LIN {X 0,Y 272.99,Z 560.234,A -85,B 0,C 180,E1 -18744.093,E2 -18744.093} C_VEL
LIN {X 0,Y 270.191,Z 556.625,A -85,B 0,C 180,E1 -18746.042,E2 -18746.042} C_VEL
LIN {X 0,Y 266.873,Z 552.939,A -85,B 0,C 180,E1 -18748.935,E2 -18748.935} C_VEL
LIN {X 0,Y 264.106,Z 550.779,A -85,B 0,C 180,E1 -18752.833,E2 -18752.833} C_VEL
LIN {X 0,Y 263.594,Z 550.284,A -85,B 0,C 180,E1 -18754.258,E2 -18754.258} C_VEL
LIN {X 0,Y 263.268,Z 551.296,A -85,B 0,C 180,E1 -18757.694,E2 -18757.694} C_VEL
LIN {X 0,Y 264.359,Z 553.676,A -85,B 0,C 180,E1 -18761.073,E2 -18761.073} C_VEL
LIN {X 0,Y 267.005,Z 559.232,A -85,B 0,C 180,E1 -18764.711,E2 -18764.711} C_VEL
LIN {X 0,Y 269.353,Z 563.234,A -85,B 0,C 180,E1 -18766.816,E2 -18766.816} C_VEL
LIN {X 0,Y 273.133,Z 570.637,A -85,B 0,C 180,E1 -18769.548,E2 -18769.548} C_VEL
LIN {X 0,Y 275.859,Z 576.586,A -85,B 0,C 180,E1 -18771.234,E2 -18771.234} C_VEL
LIN {X 0,Y 278.502,Z 582.767,A -85,B 0,C 180,E1 -18772.706,E2 -18772.706} C_VEL
LIN {X 0,Y 280.961,Z 589.169,A -85,B 0,C 180,E1 -18773.975,E2 -18773.975} C_VEL
LIN {X 0,Y 281.956,Z 602.893,A -85,B 0,C 180,E1 -18775.262,E2 -18775.262} C_VEL
LIN {X 0,Y 282.297,Z 616.005,A -85,B 0,C 180,E1 -18776.226,E2 -18776.226} C_VEL
LIN {X 0,Y 277.754,Z 659.548,A -85,B 0,C 180,E1 -18777.957,E2 -18777.957} C_VEL
LIN {X 0,Y 275.518,Z 672.942,A -85,B 0,C 180,E1 -18778.687,E2 -18778.687} C_VEL
LIN {X 0,Y 272.817,Z 685.651,A -85,B 0,C 180,E1 -18779.633,E2 -18779.633} C_VEL
LIN {X 0,Y 269.43,Z 698.811,A -85,B 0,C 180,E1 -18780.934,E2 -18780.934} C_VEL
LIN {X 0,Y 265.918,Z 710.541,A -85,B 0,C 180,E1 -18782.451,E2 -18782.451} C_VEL
LIN {X 0,Y 262.42,Z 721.186,A -85,B 0,C 180,E1 -18784.203,E2 -18784.203} C_VEL
LIN {X 0,Y 259.296,Z 730.12,A -85,B 0,C 180,E1 -18786.012,E2 -18786.012} C_VEL
LIN {X 0,Y 256.506,Z 737.614,A -85,B 0,C 180,E1 -18787.869,E2 -18787.869} C_VEL
LIN {X 0,Y 253.725,Z 745.099,A -85,B 0,C 180,E1 -18790.165,E2 -18790.165} C_VEL
LIN {X 0,Y 250.845,Z 753.157,A -85,B 0,C 180,E1 -18793.311,E2 -18793.311} C_VEL
LIN {X 0,Y 249.342,Z 760.427,A -85,B 0,C 180,E1 -18795.722,E2 -18795.722} C_VEL
LIN {X 0,Y 248.341,Z 765.333,A -85,B 0,C 180,E1 -18797.746,E2 -18797.746} C_VEL
LIN {X 0,Y 247.593,Z 770.085,A -85,B 0,C 180,E1 -18800.194,E2 -18800.194} C_VEL
LIN {X 0,Y 247.162,Z 773.704,A -85,B 0,C 180,E1 -18802.649,E2 -18802.649} C_VEL
LIN {X 0,Y 246.922,Z 776.292,A -85,B 0,C 180,E1 -18805.102,E2 -18805.102} C_VEL
LIN {X 0,Y 246.923,Z 777.505,A -85,B 0,C 180,E1 -18806.737,E2 -18806.737} C_VEL
LIN {X 0,Y 246.958,Z 778.268,A -85,B 0,C 180,E1 -18808.369,E2 -18808.369} C_VEL
LIN {X 0,Y 246.991,Z 778.625,A -85,B 0,C 180,E1 -18810,E2 -18810} C_VEL
LIN {X 0,Y 246.952,Z 778.591,A -85,B 0,C 180,E1 -18811.631,E2 -18811.631} C_VEL
LIN {X 0,Y 246.922,Z 778.159,A -85,B 0,C 180,E1 -18813.263,E2 -18813.263} C_VEL
LIN {X 0,Y 247.065,Z 776.008,A -85,B 0,C 180,E1 -18816.533,E2 -18816.533} C_VEL
LIN {X 0,Y 247.467,Z 773.301,A -85,B 0,C 180,E1 -18818.986,E2 -18818.986} C_VEL
LIN {X 0,Y 248.15,Z 769.569,A -85,B 0,C 180,E1 -18821.434,E2 -18821.434} C_VEL
LIN {X 0,Y 249.22,Z 764.704,A -85,B 0,C 180,E1 -18823.869,E2 -18823.869} C_VEL
LIN {X 0,Y 250.823,Z 758.565,A -85,B 0,C 180,E1 -18826.272,E2 -18826.272} C_VEL
LIN {X 0,Y 252.675,Z 751.27,A -85,B 0,C 180,E1 -18828.548,E2 -18828.548} C_VEL
LIN {X 0,Y 254.549,Z 743.052,A -85,B 0,C 180,E1 -18830.611,E2 -18830.611} C_VEL
LIN {X 0,Y 256.736,Z 733.463,A -85,B 0,C 180,E1 -18832.534,E2 -18832.534} C_VEL
LIN {X 0,Y 259.084,Z 722.81,A -85,B 0,C 180,E1 -18834.222,E2 -18834.222} C_VEL
LIN {X 0,Y 261.004,Z 712.424,A -85,B 0,C 180,E1 -18835.52,E2 -18835.52} C_VEL
LIN {X 0,Y 262.797,Z 701.051,A -85,B 0,C 180,E1 -18836.611,E2 -18836.611} C_VEL
LIN {X 0,Y 264.351,Z 688.267,A -85,B 0,C 180,E1 -18837.511,E2 -18837.511} C_VEL
LIN {X 0,Y 265.434,Z 675.829,A -85,B 0,C 180,E1 -18838.086,E2 -18838.086} C_VEL
LIN {X 0,Y 267.55,Z 612.058,A -85,B 0,C 180,E1 -18839.803,E2 -18839.803} C_VEL
LIN {X 0,Y 264.123,Z 582.382,A -85,B 0,C 180,E1 -18841.169,E2 -18841.169} C_VEL
LIN {X 0,Y 261.282,Z 564.651,A -85,B 0,C 180,E1 -18842.125,E2 -18842.125} C_VEL
LIN {X 0,Y 258.876,Z 558.576,A -85,B 0,C 180,E1 -18842.691,E2 -18842.691} C_VEL
LIN {X 0,Y 254.271,Z 541.842,A -85,B 0,C 180,E1 -18845.48,E2 -18845.48} C_VEL
LIN {X 0,Y 252.213,Z 535.351,A -85,B 0,C 180,E1 -18846.636,E2 -18846.636} C_VEL
LIN {X 0,Y 249.373,Z 529.876,A -85,B 0,C 180,E1 -18847.897,E2 -18847.897} C_VEL
LIN {X 0,Y 249.019,Z 528.423,A -85,B 0,C 180,E1 -18848.202,E2 -18848.202} C_VEL
LIN {X 0,Y 249.009,Z 528.461,A -85,B 0,C 180,E1 -18852.792,E2 -18852.792} C_VEL
LIN {X 0,Y 249.037,Z 528.454,A -85,B 0,C 180,E1 -18857.367,E2 -18857.367} C_VEL
LIN {X 0,Y 249.045,Z 528.46,A -85,B 0,C 180,E1 -18861.623,E2 -18861.623} C_VEL
LIN {X 0,Y 249.058,Z 528.461,A -85,B 0,C 180,E1 -18865.642,E2 -18865.642} C_VEL
LIN {X 0,Y 249.047,Z 528.44,A -85,B 0,C 180,E1 -18869.473,E2 -18869.473} C_VEL
LIN {X 0,Y 249.065,Z 528.458,A -85,B 0,C 180,E1 -18873.162,E2 -18873.162} C_VEL
LIN {X 0,Y 249.056,Z 528.434,A -85,B 0,C 180,E1 -18876.731,E2 -18876.731} C_VEL
LIN {X 0,Y 249.104,Z 528.453,A -85,B 0,C 180,E1 -18880.211,E2 -18880.211} C_VEL
LIN {X 0,Y 249.218,Z 528.409,A -85,B 0,C 180,E1 -18883.621,E2 -18883.621} C_VEL
LIN {X 0,Y 249.247,Z 528.434,A -85,B 0,C 180,E1 -18888.617,E2 -18888.617} C_VEL
LIN {X 0,Y 249.474,Z 528.375,A -85,B 0,C 180,E1 -18891.903,E2 -18891.903} C_VEL
LIN {X 0,Y 249.432,Z 528.412,A -85,B 0,C 180,E1 -18896.77,E2 -18896.77} C_VEL
LIN {X 0,Y 249.723,Z 528.342,A -85,B 0,C 180,E1 -18900,E2 -18900} C_VEL
LIN {X 0,Y 249.433,Z 528.41,A -85,B 0,C 180,E1 -18903.231,E2 -18903.231} C_VEL
LIN {X 0,Y 249.437,Z 528.393,A -85,B 0,C 180,E1 -18906.704,E2 -18906.704} C_VEL
LIN {X 0,Y 249.338,Z 528.401,A -85,B 0,C 180,E1 -18909.737,E2 -18909.737} C_VEL
LIN {X 0,Y 249.192,Z 528.424,A -85,B 0,C 180,E1 -18914.705,E2 -18914.705} C_VEL
LIN {X 0,Y 249.131,Z 528.438,A -85,B 0,C 180,E1 -18918.078,E2 -18918.078} C_VEL
LIN {X 0,Y 249.083,Z 528.449,A -85,B 0,C 180,E1 -18921.519,E2 -18921.519} C_VEL
LIN {X 0,Y 249.128,Z 528.446,A -85,B 0,C 180,E1 -18925.483,E2 -18925.483} C_VEL
LIN {X 0,Y 249.084,Z 528.44,A -85,B 0,C 180,E1 -18928.996,E2 -18928.996} C_VEL
LIN {X 0,Y 249.028,Z 528.466,A -85,B 0,C 180,E1 -18932.427,E2 -18932.427} C_VEL
LIN {X 0,Y 249.046,Z 528.46,A -85,B 0,C 180,E1 -18936.343,E2 -18936.343} C_VEL
LIN {X 0,Y 249.004,Z 528.464,A -85,B 0,C 180,E1 -18940.479,E2 -18940.479} C_VEL
LIN {X 0,Y 249.007,Z 528.47,A -85,B 0,C 180,E1 -18944.879,E2 -18944.879} C_VEL
LIN {X 0,Y 249.021,Z 528.511,A -85,B 0,C 180,E1 -18947.496,E2 -18947.496} C_VEL
LIN {X 0,Y 253.277,Z 541.471,A -85,B 0,C 180,E1 -18951.862,E2 -18951.862} C_VEL
LIN {X 0,Y 256.09,Z 551.518,A -85,B 0,C 180,E1 -18954.861,E2 -18954.861} C_VEL
LIN {X 0,Y 263.951,Z 568.494,A -85,B 0,C 180,E1 -18956.551,E2 -18956.551} C_VEL
LIN {X 0,Y 265.853,Z 573.462,A -85,B 0,C 180,E1 -18956.967,E2 -18956.967} C_VEL
LIN {X 0,Y 268.937,Z 591.166,A -85,B 0,C 180,E1 -18957.921,E2 -18957.921} C_VEL
LIN {X 0,Y 266.202,Z 662.562,A -85,B 0,C 180,E1 -18959.805,E2 -18959.805} C_VEL
LIN {X 0,Y 265.188,Z 675.566,A -85,B 0,C 180,E1 -18960.423,E2 -18960.423} C_VEL
LIN {X 0,Y 263.792,Z 688.171,A -85,B 0,C 180,E1 -18961.344,E2 -18961.344} C_VEL
LIN {X 0,Y 262.212,Z 699.557,A -85,B 0,C 180,E1 -18962.474,E2 -18962.474} C_VEL
LIN {X 0,Y 260.124,Z 711.119,A -85,B 0,C 180,E1 -18963.958,E2 -18963.958} C_VEL
LIN {X 0,Y 257.883,Z 721.5,A -85,B 0,C 180,E1 -18965.658,E2 -18965.658} C_VEL
LIN {X 0,Y 255.849,Z 729.998,A -85,B 0,C 180,E1 -18967.384,E2 -18967.384} C_VEL
LIN {X 0,Y 253.844,Z 737.814,A -85,B 0,C 180,E1 -18969.33,E2 -18969.33} C_VEL
LIN {X 0,Y 252.109,Z 744.593,A -85,B 0,C 180,E1 -18971.41,E2 -18971.41} C_VEL
LIN {X 0,Y 250.689,Z 750.647,A -85,B 0,C 180,E1 -18973.719,E2 -18973.719} C_VEL
LIN {X 0,Y 249.221,Z 755.677,A -85,B 0,C 180,E1 -18976.132,E2 -18976.132} C_VEL
LIN {X 0,Y 248.238,Z 759.549,A -85,B 0,C 180,E1 -18978.57,E2 -18978.57} C_VEL
LIN {X 0,Y 247.778,Z 761.529,A -85,B 0,C 180,E1 -18980.202,E2 -18980.202} C_VEL
LIN {X 0,Y 247.152,Z 764.272,A -85,B 0,C 180,E1 -18983.469,E2 -18983.469} C_VEL
LIN {X 0,Y 246.973,Z 765.002,A -85,B 0,C 180,E1 -18985.103,E2 -18985.103} C_VEL
LIN {X 0,Y 246.947,Z 765.341,A -85,B 0,C 180,E1 -18986.737,E2 -18986.737} C_VEL
LIN {X 0,Y 246.95,Z 765.302,A -85,B 0,C 180,E1 -18988.369,E2 -18988.369} C_VEL
LIN {X 0,Y 246.99,Z 764.874,A -85,B 0,C 180,E1 -18990,E2 -18990} C_VEL
LIN {X 0,Y 247.302,Z 762.765,A -85,B 0,C 180,E1 -18993.258,E2 -18993.258} C_VEL
LIN {X 0,Y 247.748,Z 760.11,A -85,B 0,C 180,E1 -18995.698,E2 -18995.698} C_VEL
LIN {X 0,Y 248.364,Z 756.449,A -85,B 0,C 180,E1 -18998.134,E2 -18998.134} C_VEL
LIN {X 0,Y 249.333,Z 751.675,A -85,B 0,C 180,E1 -19000.557,E2 -19000.557} C_VEL
LIN {X 0,Y 250.677,Z 745.646,A -85,B 0,C 180,E1 -19002.961,E2 -19002.961} C_VEL
LIN {X 0,Y 252.37,Z 738.111,A -85,B 0,C 180,E1 -19005.34,E2 -19005.34} C_VEL
LIN {X 0,Y 254.433,Z 728.656,A -85,B 0,C 180,E1 -19007.688,E2 -19007.688} C_VEL
LIN {X 0,Y 256.4,Z 718.895,A -85,B 0,C 180,E1 -19009.619,E2 -19009.619} C_VEL
LIN {X 0,Y 258.19,Z 709.249,A -85,B 0,C 180,E1 -19011.141,E2 -19011.141} C_VEL
LIN {X 0,Y 259.587,Z 700.508,A -85,B 0,C 180,E1 -19012.273,E2 -19012.273} C_VEL
LIN {X 0,Y 261.132,Z 689.591,A -85,B 0,C 180,E1 -19013.389,E2 -19013.389} C_VEL
LIN {X 0,Y 262.399,Z 676.059,A -85,B 0,C 180,E1 -19014.429,E2 -19014.429} C_VEL
LIN {X 0,Y 263.298,Z 663.443,A -85,B 0,C 180,E1 -19015.065,E2 -19015.065} C_VEL
LIN {X 0,Y 265.187,Z 610.796,A -85,B 0,C 180,E1 -19016.491,E2 -19016.491} C_VEL
LIN {X 0,Y 265.831,Z 588.852,A -85,B 0,C 180,E1 -19017.077,E2 -19017.077} C_VEL
LIN {X 0,Y 262.181,Z 567.297,A -85,B 0,C 180,E1 -19018.169,E2 -19018.169} C_VEL
LIN {X 0,Y 255.508,Z 551.152,A -85,B 0,C 180,E1 -19019.537,E2 -19019.537} C_VEL
LIN {X 0,Y 252.819,Z 540.961,A -85,B 0,C 180,E1 -19022.482,E2 -19022.482} C_VEL
LIN {X 0,Y 249.116,Z 528.446,A -85,B 0,C 180,E1 -19026.455,E2 -19026.455} C_VEL
LIN {X 0,Y 249.078,Z 528.446,A -85,B 0,C 180,E1 -19030.463,E2 -19030.463} C_VEL
LIN {X 0,Y 249.019,Z 528.448,A -85,B 0,C 180,E1 -19034.874,E2 -19034.874} C_VEL
LIN {X 0,Y 249.053,Z 528.465,A -85,B 0,C 180,E1 -19036.704,E2 -19036.704} C_VEL
LIN {X 0,Y 259.215,Z 557.612,A -85,B 0,C 180,E1 -19038.571,E2 -19038.571} C_VEL
LIN {X 0,Y 256.382,Z 625.461,A -85,B 0,C 180,E1 -19041.166,E2 -19041.166} C_VEL
LIN {X 0,Y 255.738,Z 638.323,A -85,B 0,C 180,E1 -19041.93,E2 -19041.93} C_VEL
LIN {X 0,Y 254.756,Z 651.647,A -85,B 0,C 180,E1 -19043.031,E2 -19043.031} C_VEL
LIN {X 0,Y 253.633,Z 664.149,A -85,B 0,C 180,E1 -19044.415,E2 -19044.415} C_VEL
LIN {X 0,Y 252.346,Z 676.451,A -85,B 0,C 180,E1 -19046.15,E2 -19046.15} C_VEL
LIN {X 0,Y 251.19,Z 687.217,A -85,B 0,C 180,E1 -19048.072,E2 -19048.072} C_VEL
LIN {X 0,Y 250.005,Z 691.571,A -85,B 0,C 180,E1 -19048.949,E2 -19048.949} C_VEL
LIN {X 0,Y 246.343,Z 698.223,A -85,B 0,C 180,E1 -19050.431,E2 -19050.431} C_VEL
LIN {X 0,Y 242.767,Z 704.382,A -85,B 0,C 180,E1 -19052.06,E2 -19052.06} C_VEL
LIN {X 0,Y 241.73,Z 707.892,A -85,B 0,C 180,E1 -19053.148,E2 -19053.148} C_VEL
LIN {X 0,Y 241.207,Z 713.595,A -85,B 0,C 180,E1 -19055.206,E2 -19055.206} C_VEL
LIN {X 0,Y 240.618,Z 719.237,A -85,B 0,C 180,E1 -19057.684,E2 -19057.684} C_VEL
LIN {X 0,Y 240.293,Z 723.943,A -85,B 0,C 180,E1 -19060.345,E2 -19060.345} C_VEL
LIN {X 0,Y 240.205,Z 727.388,A -85,B 0,C 180,E1 -19062.987,E2 -19062.987} C_VEL
LIN {X 0,Y 240.325,Z 729.1,A -85,B 0,C 180,E1 -19064.801,E2 -19064.801} C_VEL
LIN {X 0,Y 240.548,Z 730.266,A -85,B 0,C 180,E1 -19066.483,E2 -19066.483} C_VEL
LIN {X 0,Y 240.898,Z 731.008,A -85,B 0,C 180,E1 -19068.216,E2 -19068.216} C_VEL
LIN {X 0,Y 241.855,Z 731.244,A -85,B 0,C 180,E1 -19071.105,E2 -19071.105} C_VEL
LIN {X 0,Y 242.816,Z 730.604,A -85,B 0,C 180,E1 -19073.351,E2 -19073.351} C_VEL
LIN {X 0,Y 243.776,Z 729.566,A -85,B 0,C 180,E1 -19075.038,E2 -19075.038} C_VEL
LIN {X 0,Y 246.085,Z 726.341,A -85,B 0,C 180,E1 -19078.28,E2 -19078.28} C_VEL
LIN {X 0,Y 248.337,Z 722.512,A -85,B 0,C 180,E1 -19080.81,E2 -19080.81} C_VEL
LIN {X 0,Y 250.903,Z 717.616,A -85,B 0,C 180,E1 -19083.211,E2 -19083.211} C_VEL
LIN {X 0,Y 253.556,Z 712.049,A -85,B 0,C 180,E1 -19085.347,E2 -19085.347} C_VEL
LIN {X 0,Y 256.664,Z 705.116,A -85,B 0,C 180,E1 -19087.473,E2 -19087.473} C_VEL
LIN {X 0,Y 260.263,Z 695.935,A -85,B 0,C 180,E1 -19089.716,E2 -19089.716} C_VEL
LIN {X 0,Y 263.627,Z 686.39,A -85,B 0,C 180,E1 -19091.533,E2 -19091.533} C_VEL
LIN {X 0,Y 266.924,Z 675.627,A -85,B 0,C 180,E1 -19093.185,E2 -19093.185} C_VEL
LIN {X 0,Y 270.017,Z 663.83,A -85,B 0,C 180,E1 -19094.6,E2 -19094.6} C_VEL
LIN {X 0,Y 272.46,Z 651.925,A -85,B 0,C 180,E1 -19095.714,E2 -19095.714} C_VEL
LIN {X 0,Y 274.515,Z 638.818,A -85,B 0,C 180,E1 -19096.643,E2 -19096.643} C_VEL
LIN {X 0,Y 276.515,Z 620.559,A -85,B 0,C 180,E1 -19097.519,E2 -19097.519} C_VEL
LIN {X 0,Y 280.862,Z 583.373,A -85,B 0,C 180,E1 -19098.983,E2 -19098.983} C_VEL
LIN {X 0,Y 277.859,Z 577.693,A -85,B 0,C 180,E1 -19100.43,E2 -19100.43} C_VEL
LIN {X 0,Y 274.432,Z 572.112,A -85,B 0,C 180,E1 -19102.221,E2 -19102.221} C_VEL
LIN {X 0,Y 271.179,Z 567.198,A -85,B 0,C 180,E1 -19104.186,E2 -19104.186} C_VEL
LIN {X 0,Y 268.152,Z 563.271,A -85,B 0,C 180,E1 -19106.357,E2 -19106.357} C_VEL
LIN {X 0,Y 265.242,Z 559.819,A -85,B 0,C 180,E1 -19109.03,E2 -19109.03} C_VEL
LIN {X 0,Y 262.508,Z 557.611,A -85,B 0,C 180,E1 -19113.059,E2 -19113.059} C_VEL
LIN {X 0,Y 262.098,Z 557.203,A -85,B 0,C 180,E1 -19114.27,E2 -19114.27} C_VEL
LIN {X 0,Y 261.741,Z 558.144,A -85,B 0,C 180,E1 -19117.454,E2 -19117.454} C_VEL
LIN {X 0,Y 262.545,Z 560.201,A -85,B 0,C 180,E1 -19120.455,E2 -19120.455} C_VEL
LIN {X 0,Y 263.676,Z 562.983,A -85,B 0,C 180,E1 -19122.571,E2 -19122.571} C_VEL
LIN {X 0,Y 266.928,Z 569.26,A -85,B 0,C 180,E1 -19126.2,E2 -19126.2} C_VEL
LIN {X 0,Y 270.377,Z 576.507,A -85,B 0,C 180,E1 -19128.921,E2 -19128.921} C_VEL
LIN {X 0,Y 273.124,Z 582.914,A -85,B 0,C 180,E1 -19130.764,E2 -19130.764} C_VEL
LIN {X 0,Y 276.12,Z 590.349,A -85,B 0,C 180,E1 -19132.51,E2 -19132.51} C_VEL
LIN {X 0,Y 277.009,Z 593.418,A -85,B 0,C 180,E1 -19133.072,E2 -19133.072} C_VEL
LIN {X 0,Y 277.845,Z 607.865,A -85,B 0,C 180,E1 -19134.425,E2 -19134.425} C_VEL
LIN {X 0,Y 277.751,Z 618.425,A -85,B 0,C 180,E1 -19135.169,E2 -19135.169} C_VEL
LIN {X 0,Y 273.212,Z 659.053,A -85,B 0,C 180,E1 -19136.81,E2 -19136.81} C_VEL
LIN {X 0,Y 270.87,Z 672.342,A -85,B 0,C 180,E1 -19137.538,E2 -19137.538} C_VEL
LIN {X 0,Y 268.261,Z 683.948,A -85,B 0,C 180,E1 -19138.402,E2 -19138.402} C_VEL
LIN {X 0,Y 264.647,Z 697.137,A -85,B 0,C 180,E1 -19139.698,E2 -19139.698} C_VEL
LIN {X 0,Y 260.928,Z 709.059,A -85,B 0,C 180,E1 -19141.22,E2 -19141.22} C_VEL
LIN {X 0,Y 257.566,Z 718.845,A -85,B 0,C 180,E1 -19142.804,E2 -19142.804} C_VEL
LIN {X 0,Y 253.548,Z 729.603,A -85,B 0,C 180,E1 -19144.995,E2 -19144.995} C_VEL
LIN {X 0,Y 249.998,Z 738.361,A -85,B 0,C 180,E1 -19147.261,E2 -19147.261} C_VEL
LIN {X 0,Y 246.656,Z 746.661,A -85,B 0,C 180,E1 -19150.007,E2 -19150.007} C_VEL
LIN {X 0,Y 244.02,Z 753.185,A -85,B 0,C 180,E1 -19152.83,E2 -19152.83} C_VEL
LIN {X 0,Y 241.954,Z 762.239,A -85,B 0,C 180,E1 -19156.135,E2 -19156.135} C_VEL
LIN {X 0,Y 240.799,Z 768.416,A -85,B 0,C 180,E1 -19159.064,E2 -19159.064} C_VEL
LIN {X 0,Y 240.212,Z 772.409,A -85,B 0,C 180,E1 -19161.588,E2 -19161.588} C_VEL
LIN {X 0,Y 239.996,Z 774.455,A -85,B 0,C 180,E1 -19163.273,E2 -19163.273} C_VEL
LIN {X 0,Y 239.839,Z 776.177,A -85,B 0,C 180,E1 -19165.071,E2 -19165.071} C_VEL
LIN {X 0,Y 239.824,Z 777.297,A -85,B 0,C 180,E1 -19166.64,E2 -19166.64} C_VEL
LIN {X 0,Y 239.867,Z 778.07,A -85,B 0,C 180,E1 -19168.321,E2 -19168.321} C_VEL
LIN {X 0,Y 239.9,Z 778.432,A -85,B 0,C 180,E1 -19170,E2 -19170} C_VEL
LIN {X 0,Y 239.862,Z 778.402,A -85,B 0,C 180,E1 -19171.679,E2 -19171.679} C_VEL
LIN {X 0,Y 239.824,Z 777.978,A -85,B 0,C 180,E1 -19173.36,E2 -19173.36} C_VEL
LIN {X 0,Y 239.844,Z 777.109,A -85,B 0,C 180,E1 -19175.043,E2 -19175.043} C_VEL
LIN {X 0,Y 239.989,Z 775.839,A -85,B 0,C 180,E1 -19176.727,E2 -19176.727} C_VEL
LIN {X 0,Y 240.423,Z 773.143,A -85,B 0,C 180,E1 -19179.252,E2 -19179.252} C_VEL
LIN {X 0,Y 241.167,Z 769.423,A -85,B 0,C 180,E1 -19181.77,E2 -19181.77} C_VEL
LIN {X 0,Y 242.301,Z 764.57,A -85,B 0,C 180,E1 -19184.273,E2 -19184.273} C_VEL
LIN {X 0,Y 243.983,Z 758.445,A -85,B 0,C 180,E1 -19186.741,E2 -19186.741} C_VEL
LIN {X 0,Y 245.851,Z 751.48,A -85,B 0,C 180,E1 -19188.985,E2 -19188.985} C_VEL
LIN {X 0,Y 247.885,Z 742.978,A -85,B 0,C 180,E1 -19191.191,E2 -19191.191} C_VEL
LIN {X 0,Y 250.201,Z 733.413,A -85,B 0,C 180,E1 -19193.156,E2 -19193.156} C_VEL
LIN {X 0,Y 252.61,Z 722.793,A -85,B 0,C 180,E1 -19194.884,E2 -19194.884} C_VEL
LIN {X 0,Y 254.621,Z 712.468,A -85,B 0,C 180,E1 -19196.207,E2 -19196.207} C_VEL
LIN {X 0,Y 256.627,Z 700.06,A -85,B 0,C 180,E1 -19197.414,E2 -19197.414} C_VEL
LIN {X 0,Y 258.289,Z 686.996,A -85,B 0,C 180,E1 -19198.324,E2 -19198.324} C_VEL
LIN {X 0,Y 259.349,Z 673.611,A -85,B 0,C 180,E1 -19198.916,E2 -19198.916} C_VEL
LIN {X 0,Y 261.477,Z 613.223,A -85,B 0,C 180,E1 -19200.557,E2 -19200.557} C_VEL
LIN {X 0,Y 258.243,Z 584.392,A -85,B 0,C 180,E1 -19201.923,E2 -19201.923} C_VEL
LIN {X 0,Y 255.65,Z 567.616,A -85,B 0,C 180,E1 -19202.849,E2 -19202.849} C_VEL
LIN {X 0,Y 252.033,Z 558.209,A -85,B 0,C 180,E1 -19203.763,E2 -19203.763} C_VEL
LIN {X 0,Y 247.176,Z 540.889,A -85,B 0,C 180,E1 -19206.845,E2 -19206.845} C_VEL
LIN {X 0,Y 245.96,Z 537.781,A -85,B 0,C 180,E1 -19207.469,E2 -19207.469} C_VEL
LIN {X 0,Y 242.282,Z 530.723,A -85,B 0,C 180,E1 -19209.207,E2 -19209.207} C_VEL
LIN {X 0,Y 241.943,Z 529.312,A -85,B 0,C 180,E1 -19209.533,E2 -19209.533} C_VEL
LIN {X 0,Y 241.935,Z 529.338,A -85,B 0,C 180,E1 -19213.429,E2 -19213.429} C_VEL
LIN {X 0,Y 241.973,Z 529.343,A -85,B 0,C 180,E1 -19216.56,E2 -19216.56} C_VEL
LIN {X 0,Y 241.978,Z 529.344,A -85,B 0,C 180,E1 -19220.285,E2 -19220.285} C_VEL
LIN {X 0,Y 242.033,Z 529.323,A -85,B 0,C 180,E1 -19224.497,E2 -19224.497} C_VEL
LIN {X 0,Y 241.971,Z 529.324,A -85,B 0,C 180,E1 -19228.48,E2 -19228.48} C_VEL
LIN {X 0,Y 242.003,Z 529.339,A -85,B 0,C 180,E1 -19232.312,E2 -19232.312} C_VEL
LIN {X 0,Y 242.036,Z 529.306,A -85,B 0,C 180,E1 -19236.014,E2 -19236.014} C_VEL
LIN {X 0,Y 242.031,Z 529.336,A -85,B 0,C 180,E1 -19239.608,E2 -19239.608} C_VEL
LIN {X 0,Y 242.158,Z 529.288,A -85,B 0,C 180,E1 -19243.278,E2 -19243.278} C_VEL
LIN {X 0,Y 242.181,Z 529.317,A -85,B 0,C 180,E1 -19248.28,E2 -19248.28} C_VEL
LIN {X 0,Y 242.421,Z 529.253,A -85,B 0,C 180,E1 -19251.666,E2 -19251.666} C_VEL
LIN {X 0,Y 242.256,Z 529.305,A -85,B 0,C 180,E1 -19255.007,E2 -19255.007} C_VEL
LIN {X 0,Y 242.632,Z 529.238,A -85,B 0,C 180,E1 -19258.341,E2 -19258.341} C_VEL
LIN {X 0,Y 242.632,Z 529.236,A -85,B 0,C 180,E1 -19261.66,E2 -19261.66} C_VEL
LIN {X 0,Y 242.418,Z 529.267,A -85,B 0,C 180,E1 -19266.676,E2 -19266.676} C_VEL
LIN {X 0,Y 242.263,Z 529.286,A -85,B 0,C 180,E1 -19270.024,E2 -19270.024} C_VEL
LIN {X 0,Y 242.152,Z 529.296,A -85,B 0,C 180,E1 -19275.142,E2 -19275.142} C_VEL
LIN {X 0,Y 242.067,Z 529.326,A -85,B 0,C 180,E1 -19278.625,E2 -19278.625} C_VEL
LIN {X 0,Y 242.009,Z 529.32,A -85,B 0,C 180,E1 -19282.181,E2 -19282.181} C_VEL
LIN {X 0,Y 242.064,Z 529.331,A -85,B 0,C 180,E1 -19285.839,E2 -19285.839} C_VEL
LIN {X 0,Y 242.029,Z 529.317,A -85,B 0,C 180,E1 -19289.581,E2 -19289.581} C_VEL
LIN {X 0,Y 241.978,Z 529.338,A -85,B 0,C 180,E1 -19293.494,E2 -19293.494} C_VEL
LIN {X 0,Y 241.988,Z 529.346,A -85,B 0,C 180,E1 -19297.583,E2 -19297.583} C_VEL
LIN {X 0,Y 241.938,Z 529.355,A -85,B 0,C 180,E1 -19301.923,E2 -19301.923} C_VEL
LIN {X 0,Y 241.953,Z 529.487,A -85,B 0,C 180,E1 -19306.339,E2 -19306.339} C_VEL
LIN {X 0,Y 245.448,Z 539.786,A -85,B 0,C 180,E1 -19309.991,E2 -19309.991} C_VEL
LIN {X 0,Y 248.246,Z 548.984,A -85,B 0,C 180,E1 -19312.988,E2 -19312.988} C_VEL
LIN {X 0,Y 249.025,Z 551.686,A -85,B 0,C 180,E1 -19313.757,E2 -19313.757} C_VEL
LIN {X 0,Y 256.527,Z 567.423,A -85,B 0,C 180,E1 -19315.454,E2 -19315.454} C_VEL
LIN {X 0,Y 260.054,Z 575.918,A -85,B 0,C 180,E1 -19316.242,E2 -19316.242} C_VEL
LIN {X 0,Y 262.837,Z 592.295,A -85,B 0,C 180,E1 -19317.151,E2 -19317.151} C_VEL
LIN {X 0,Y 260.022,Z 663.023,A -85,B 0,C 180,E1 -19319.058,E2 -19319.058} C_VEL
LIN {X 0,Y 258.944,Z 676.006,A -85,B 0,C 180,E1 -19319.692,E2 -19319.692} C_VEL
LIN {X 0,Y 257.595,Z 688.014,A -85,B 0,C 180,E1 -19320.588,E2 -19320.588} C_VEL
LIN {X 0,Y 255.92,Z 699.316,A -85,B 0,C 180,E1 -19321.717,E2 -19321.717} C_VEL
LIN {X 0,Y 254.04,Z 709.803,A -85,B 0,C 180,E1 -19323.063,E2 -19323.063} C_VEL
LIN {X 0,Y 251.675,Z 720.483,A -85,B 0,C 180,E1 -19324.796,E2 -19324.796} C_VEL
LIN {X 0,Y 249.285,Z 730.052,A -85,B 0,C 180,E1 -19326.754,E2 -19326.754} C_VEL
LIN {X 0,Y 247.191,Z 737.892,A -85,B 0,C 180,E1 -19328.747,E2 -19328.747} C_VEL
LIN {X 0,Y 245.256,Z 745.115,A -85,B 0,C 180,E1 -19331.023,E2 -19331.023} C_VEL
LIN {X 0,Y 243.852,Z 750.763,A -85,B 0,C 180,E1 -19333.25,E2 -19333.25} C_VEL
LIN {X 0,Y 242.3,Z 755.813,A -85,B 0,C 180,E1 -19335.727,E2 -19335.727} C_VEL
LIN {X 0,Y 241.245,Z 759.7,A -85,B 0,C 180,E1 -19338.234,E2 -19338.234} C_VEL
LIN {X 0,Y 240.745,Z 761.688,A -85,B 0,C 180,E1 -19339.913,E2 -19339.913} C_VEL
LIN {X 0,Y 240.36,Z 763.265,A -85,B 0,C 180,E1 -19341.594,E2 -19341.594} C_VEL
LIN {X 0,Y 240.076,Z 764.444,A -85,B 0,C 180,E1 -19343.276,E2 -19343.276} C_VEL
LIN {X 0,Y 239.85,Z 765.529,A -85,B 0,C 180,E1 -19346.64,E2 -19346.64} C_VEL
LIN {X 0,Y 239.862,Z 765.495,A -85,B 0,C 180,E1 -19348.321,E2 -19348.321} C_VEL
LIN {X 0,Y 239.898,Z 765.077,A -85,B 0,C 180,E1 -19350,E2 -19350} C_VEL
LIN {X 0,Y 240.224,Z 762.982,A -85,B 0,C 180,E1 -19353.354,E2 -19353.354} C_VEL
LIN {X 0,Y 240.699,Z 760.34,A -85,B 0,C 180,E1 -19355.865,E2 -19355.865} C_VEL
LIN {X 0,Y 241.337,Z 756.692,A -85,B 0,C 180,E1 -19358.372,E2 -19358.372} C_VEL
LIN {X 0,Y 242.367,Z 751.93,A -85,B 0,C 180,E1 -19360.864,E2 -19360.864} C_VEL
LIN {X 0,Y 243.762,Z 745.917,A -85,B 0,C 180,E1 -19363.335,E2 -19363.335} C_VEL
LIN {X 0,Y 245.549,Z 738.406,A -85,B 0,C 180,E1 -19365.777,E2 -19365.777} C_VEL
LIN {X 0,Y 247.684,Z 728.971,A -85,B 0,C 180,E1 -19368.187,E2 -19368.187} C_VEL
LIN {X 0,Y 249.742,Z 719.241,A -85,B 0,C 180,E1 -19370.165,E2 -19370.165} C_VEL
LIN {X 0,Y 251.858,Z 708.257,A -85,B 0,C 180,E1 -19371.914,E2 -19371.914} C_VEL
LIN {X 0,Y 253.502,Z 697.557,A -85,B 0,C 180,E1 -19373.269,E2 -19373.269} C_VEL
LIN {X 0,Y 255.139,Z 685.78,A -85,B 0,C 180,E1 -19374.404,E2 -19374.404} C_VEL
LIN {X 0,Y 256.275,Z 673.355,A -85,B 0,C 180,E1 -19375.282,E2 -19375.282} C_VEL
LIN {X 0,Y 257.092,Z 660.341,A -85,B 0,C 180,E1 -19375.879,E2 -19375.879} C_VEL
LIN {X 0,Y 259.568,Z 589.737,A -85,B 0,C 180,E1 -19377.794,E2 -19377.794} C_VEL
LIN {X 0,Y 256.281,Z 569.876,A -85,B 0,C 180,E1 -19378.83,E2 -19378.83} C_VEL
LIN {X 0,Y 249.913,Z 554.576,A -85,B 0,C 180,E1 -19380.179,E2 -19380.179} C_VEL
LIN {X 0,Y 248.374,Z 551.252,A -85,B 0,C 180,E1 -19380.527,E2 -19380.527} C_VEL
LIN {X 0,Y 245.37,Z 540.268,A -85,B 0,C 180,E1 -19383.835,E2 -19383.835} C_VEL
LIN {X 0,Y 242.531,Z 531.085,A -85,B 0,C 180,E1 -19386.831,E2 -19386.831} C_VEL
LIN {X 0,Y 242.045,Z 529.329,A -85,B 0,C 180,E1 -19387.444,E2 -19387.444} C_VEL
LIN {X 0,Y 241.985,Z 529.34,A -85,B 0,C 180,E1 -19391.911,E2 -19391.911} C_VEL
LIN {X 0,Y 241.996,Z 529.326,A -85,B 0,C 180,E1 -19396.22,E2 -19396.22} C_VEL
LIN {X 0,Y 252.286,Z 558.661,A -85,B 0,C 180,E1 -19398.196,E2 -19398.196} C_VEL
LIN {X 0,Y 249.369,Z 626.904,A -85,B 0,C 180,E1 -19400.905,E2 -19400.905} C_VEL
LIN {X 0,Y 248.55,Z 641.62,A -85,B 0,C 180,E1 -19401.845,E2 -19401.845} C_VEL
LIN {X 0,Y 247.487,Z 654.999,A -85,B 0,C 180,E1 -19403.068,E2 -19403.068} C_VEL
LIN {X 0,Y 246.411,Z 666.79,A -85,B 0,C 180,E1 -19404.47,E2 -19404.47} C_VEL
LIN {X 0,Y 245.127,Z 678.554,A -85,B 0,C 180,E1 -19406.246,E2 -19406.246} C_VEL
LIN {X 0,Y 243.891,Z 689.32,A -85,B 0,C 180,E1 -19408.271,E2 -19408.271} C_VEL
LIN {X 0,Y 242.731,Z 698.866,A -85,B 0,C 180,E1 -19410.513,E2 -19410.513} C_VEL
LIN {X 0,Y 241.73,Z 707.892,A -85,B 0,C 180,E1 -19413.148,E2 -19413.148} C_VEL
LIN {X 0,Y 240.737,Z 711.274,A -85,B 0,C 180,E1 -19414.274,E2 -19414.274} C_VEL
LIN {X 0,Y 237.396,Z 716.201,A -85,B 0,C 180,E1 -19416.175,E2 -19416.175} C_VEL
LIN {X 0,Y 234.126,Z 720.461,A -85,B 0,C 180,E1 -19418.219,E2 -19418.219} C_VEL
LIN {X 0,Y 233.273,Z 722.804,A -85,B 0,C 180,E1 -19419.543,E2 -19419.543} C_VEL
LIN {X 0,Y 233.085,Z 726.957,A -85,B 0,C 180,E1 -19422.451,E2 -19422.451} C_VEL
LIN {X 0,Y 233.204,Z 729.252,A -85,B 0,C 180,E1 -19424.655,E2 -19424.655} C_VEL
LIN {X 0,Y 233.712,Z 731.301,A -85,B 0,C 180,E1 -19427.848,E2 -19427.848} C_VEL
LIN {X 0,Y 234.76,Z 731.962,A -85,B 0,C 180,E1 -19431.077,E2 -19431.077} C_VEL
LIN {X 0,Y 235.629,Z 731.589,A -85,B 0,C 180,E1 -19433.147,E2 -19433.147} C_VEL
LIN {X 0,Y 236.599,Z 730.821,A -85,B 0,C 180,E1 -19434.887,E2 -19434.887} C_VEL
LIN {X 0,Y 237.726,Z 729.639,A -85,B 0,C 180,E1 -19436.61,E2 -19436.61} C_VEL
LIN {X 0,Y 239.728,Z 726.97,A -85,B 0,C 180,E1 -19439.183,E2 -19439.183} C_VEL
LIN {X 0,Y 242.087,Z 723.287,A -85,B 0,C 180,E1 -19441.663,E2 -19441.663} C_VEL
LIN {X 0,Y 244.858,Z 718.468,A -85,B 0,C 180,E1 -19444.114,E2 -19444.114} C_VEL
LIN {X 0,Y 248.055,Z 712.336,A -85,B 0,C 180,E1 -19446.507,E2 -19446.507} C_VEL
LIN {X 0,Y 251.649,Z 704.671,A -85,B 0,C 180,E1 -19448.835,E2 -19448.835} C_VEL
LIN {X 0,Y 254.867,Z 696.98,A -85,B 0,C 180,E1 -19450.727,E2 -19450.727} C_VEL
LIN {X 0,Y 258.446,Z 687.639,A -85,B 0,C 180,E1 -19452.565,E2 -19452.565} C_VEL
LIN {X 0,Y 261.954,Z 676.868,A -85,B 0,C 180,E1 -19454.245,E2 -19454.245} C_VEL
LIN {X 0,Y 265.381,Z 664.493,A -85,B 0,C 180,E1 -19455.75,E2 -19455.75} C_VEL
LIN {X 0,Y 268.135,Z 651.87,A -85,B 0,C 180,E1 -19456.953,E2 -19456.953} C_VEL
LIN {X 0,Y 270.358,Z 638.578,A -85,B 0,C 180,E1 -19457.882,E2 -19457.882} C_VEL
LIN {X 0,Y 272.786,Z 617.726,A -85,B 0,C 180,E1 -19458.848,E2 -19458.848} C_VEL
LIN {X 0,Y 276.643,Z 586.919,A -85,B 0,C 180,E1 -19460.075,E2 -19460.075} C_VEL
LIN {X 0,Y 273.069,Z 580.296,A -85,B 0,C 180,E1 -19461.983,E2 -19461.983} C_VEL
LIN {X 0,Y 269.543,Z 574.7,A -85,B 0,C 180,E1 -19464.138,E2 -19464.138} C_VEL
LIN {X 0,Y 266.035,Z 569.82,A -85,B 0,C 180,E1 -19466.76,E2 -19466.76} C_VEL
LIN {X 0,Y 263.406,Z 566.587,A -85,B 0,C 180,E1 -19469.357,E2 -19469.357} C_VEL
LIN {X 0,Y 260.87,Z 564.439,A -85,B 0,C 180,E1 -19473.37,E2 -19473.37} C_VEL
LIN {X 0,Y 260.423,Z 564.248,A -85,B 0,C 180,E1 -19475.018,E2 -19475.018} C_VEL
LIN {X 0,Y 260.358,Z 565.681,A -85,B 0,C 180,E1 -19478.483,E2 -19478.483} C_VEL
LIN {X 0,Y 261.159,Z 567.66,A -85,B 0,C 180,E1 -19480.825,E2 -19480.825} C_VEL
LIN {X 0,Y 263.691,Z 573.596,A -85,B 0,C 180,E1 -19484.62,E2 -19484.62} C_VEL
LIN {X 0,Y 264.865,Z 575.972,A -85,B 0,C 180,E1 -19485.833,E2 -19485.833} C_VEL
LIN {X 0,Y 267.706,Z 582.386,A -85,B 0,C 180,E1 -19488.284,E2 -19488.284} C_VEL
LIN {X 0,Y 270.055,Z 588.14,A -85,B 0,C 180,E1 -19489.981,E2 -19489.981} C_VEL
LIN {X 0,Y 272.71,Z 595.265,A -85,B 0,C 180,E1 -19491.713,E2 -19491.713} C_VEL
LIN {X 0,Y 273.267,Z 597.625,A -85,B 0,C 180,E1 -19492.119,E2 -19492.119} C_VEL
LIN {X 0,Y 273.688,Z 610.926,A -85,B 0,C 180,E1 -19493.388,E2 -19493.388} C_VEL
LIN {X 0,Y 273.537,Z 619.695,A -85,B 0,C 180,E1 -19494.01,E2 -19494.01} C_VEL
LIN {X 0,Y 268.795,Z 658.983,A -85,B 0,C 180,E1 -19495.627,E2 -19495.627} C_VEL
LIN {X 0,Y 266.089,Z 673.025,A -85,B 0,C 180,E1 -19496.427,E2 -19496.427} C_VEL
LIN {X 0,Y 262.91,Z 686.042,A -85,B 0,C 180,E1 -19497.455,E2 -19497.455} C_VEL
LIN {X 0,Y 259.176,Z 698.695,A -85,B 0,C 180,E1 -19498.762,E2 -19498.762} C_VEL
LIN {X 0,Y 255.277,Z 710.077,A -85,B 0,C 180,E1 -19500.294,E2 -19500.294} C_VEL
LIN {X 0,Y 252.129,Z 718.525,A -85,B 0,C 180,E1 -19501.715,E2 -19501.715} C_VEL
LIN {X 0,Y 247.877,Z 729.21,A -85,B 0,C 180,E1 -19503.931,E2 -19503.931} C_VEL
LIN {X 0,Y 244.095,Z 737.884,A -85,B 0,C 180,E1 -19506.229,E2 -19506.229} C_VEL
LIN {X 0,Y 240.466,Z 746.073,A -85,B 0,C 180,E1 -19509.022,E2 -19509.022} C_VEL
LIN {X 0,Y 237.605,Z 752.579,A -85,B 0,C 180,E1 -19511.907,E2 -19511.907} C_VEL
LIN {X 0,Y 236.734,Z 754.613,A -85,B 0,C 180,E1 -19512.953,E2 -19512.953} C_VEL
LIN {X 0,Y 235.295,Z 760.98,A -85,B 0,C 180,E1 -19515.293,E2 -19515.293} C_VEL
LIN {X 0,Y 234.086,Z 766.568,A -85,B 0,C 180,E1 -19517.868,E2 -19517.868} C_VEL
LIN {X 0,Y 233.319,Z 770.946,A -85,B 0,C 180,E1 -19520.464,E2 -19520.464} C_VEL
LIN {X 0,Y 232.924,Z 774.236,A -85,B 0,C 180,E1 -19523.068,E2 -19523.068} C_VEL
LIN {X 0,Y 232.761,Z 776.148,A -85,B 0,C 180,E1 -19525.14,E2 -19525.14} C_VEL
LIN {X 0,Y 232.779,Z 777.871,A -85,B 0,C 180,E1 -19528.27,E2 -19528.27} C_VEL
LIN {X 0,Y 232.81,Z 778.239,A -85,B 0,C 180,E1 -19530,E2 -19530} C_VEL
LIN {X 0,Y 232.774,Z 778.214,A -85,B 0,C 180,E1 -19531.73,E2 -19531.73} C_VEL
LIN {X 0,Y 232.761,Z 777.148,A -85,B 0,C 180,E1 -19534.861,E2 -19534.861} C_VEL
LIN {X 0,Y 232.916,Z 775.671,A -85,B 0,C 180,E1 -19536.932,E2 -19536.932} C_VEL
LIN {X 0,Y 233.399,Z 772.986,A -85,B 0,C 180,E1 -19539.533,E2 -19539.533} C_VEL
LIN {X 0,Y 234.178,Z 769.276,A -85,B 0,C 180,E1 -19542.127,E2 -19542.127} C_VEL
LIN {X 0,Y 235.403,Z 764.437,A -85,B 0,C 180,E1 -19544.7,E2 -19544.7} C_VEL
LIN {X 0,Y 237.158,Z 758.326,A -85,B 0,C 180,E1 -19547.238,E2 -19547.238} C_VEL
LIN {X 0,Y 239.319,Z 750.481,A -85,B 0,C 180,E1 -19549.808,E2 -19549.808} C_VEL
LIN {X 0,Y 241.687,Z 741.137,A -85,B 0,C 180,E1 -19552.211,E2 -19552.211} C_VEL
LIN {X 0,Y 244.244,Z 731.242,A -85,B 0,C 180,E1 -19554.206,E2 -19554.206} C_VEL
LIN {X 0,Y 246.759,Z 720.028,A -85,B 0,C 180,E1 -19555.969,E2 -19555.969} C_VEL
LIN {X 0,Y 248.849,Z 709.044,A -85,B 0,C 180,E1 -19557.317,E2 -19557.317} C_VEL
LIN {X 0,Y 250.835,Z 696.797,A -85,B 0,C 180,E1 -19558.444,E2 -19558.444} C_VEL
LIN {X 0,Y 252.385,Z 683.81,A -85,B 0,C 180,E1 -19559.277,E2 -19559.277} C_VEL
LIN {X 0,Y 253.325,Z 671.397,A -85,B 0,C 180,E1 -19559.786,E2 -19559.786} C_VEL
LIN {X 0,Y 255.433,Z 613.963,A -85,B 0,C 180,E1 -19561.364,E2 -19561.364} C_VEL
LIN {X 0,Y 252.114,Z 584.183,A -85,B 0,C 180,E1 -19562.831,E2 -19562.831} C_VEL
LIN {X 0,Y 250.002,Z 570.393,A -85,B 0,C 180,E1 -19563.622,E2 -19563.622} C_VEL
LIN {X 0,Y 245.275,Z 558.328,A -85,B 0,C 180,E1 -19564.831,E2 -19564.831} C_VEL
LIN {X 0,Y 241.434,Z 543.99,A -85,B 0,C 180,E1 -19567.513,E2 -19567.513} C_VEL
LIN {X 0,Y 236.446,Z 533.803,A -85,B 0,C 180,E1 -19569.99,E2 -19569.99} C_VEL
LIN {X 0,Y 235.003,Z 530.88,A -85,B 0,C 180,E1 -19570.757,E2 -19570.757} C_VEL
LIN {X 0,Y 234.9,Z 530.215,A -85,B 0,C 180,E1 -19570.947,E2 -19570.947} C_VEL
LIN {X 0,Y 234.926,Z 530.225,A -85,B 0,C 180,E1 -19575.886,E2 -19575.886} C_VEL
LIN {X 0,Y 234.908,Z 530.21,A -85,B 0,C 180,E1 -19578.838,E2 -19578.838} C_VEL
LIN {X 0,Y 234.952,Z 530.219,A -85,B 0,C 180,E1 -19581.085,E2 -19581.085} C_VEL
LIN {X 0,Y 234.957,Z 530.213,A -85,B 0,C 180,E1 -19585.367,E2 -19585.367} C_VEL
LIN {X 0,Y 234.965,Z 530.196,A -85,B 0,C 180,E1 -19590.157,E2 -19590.157} C_VEL
LIN {X 0,Y 234.99,Z 530.205,A -85,B 0,C 180,E1 -19593.793,E2 -19593.793} C_VEL
LIN {X 0,Y 234.993,Z 530.21,A -85,B 0,C 180,E1 -19598.968,E2 -19598.968} C_VEL
LIN {X 0,Y 235.091,Z 530.169,A -85,B 0,C 180,E1 -19603.06,E2 -19603.06} C_VEL
LIN {X 0,Y 235.141,Z 530.194,A -85,B 0,C 180,E1 -19607.924,E2 -19607.924} C_VEL
LIN {X 0,Y 235.371,Z 530.131,A -85,B 0,C 180,E1 -19611.414,E2 -19611.414} C_VEL
LIN {X 0,Y 235.398,Z 530.137,A -85,B 0,C 180,E1 -19613.142,E2 -19613.142} C_VEL
LIN {X 0,Y 235.591,Z 530.115,A -85,B 0,C 180,E1 -19618.291,E2 -19618.291} C_VEL
LIN {X 0,Y 235.592,Z 530.113,A -85,B 0,C 180,E1 -19621.71,E2 -19621.71} C_VEL
LIN {X 0,Y 235.369,Z 530.142,A -85,B 0,C 180,E1 -19626.86,E2 -19626.86} C_VEL
LIN {X 0,Y 235.21,Z 530.168,A -85,B 0,C 180,E1 -19630.328,E2 -19630.328} C_VEL
LIN {X 0,Y 235.103,Z 530.17,A -85,B 0,C 180,E1 -19635.608,E2 -19635.608} C_VEL
LIN {X 0,Y 235.004,Z 530.21,A -85,B 0,C 180,E1 -19639.207,E2 -19639.207} C_VEL
LIN {X 0,Y 234.957,Z 530.193,A -85,B 0,C 180,E1 -19642.884,E2 -19642.884} C_VEL
LIN {X 0,Y 234.968,Z 530.218,A -85,B 0,C 180,E1 -19646.658,E2 -19646.658} C_VEL
LIN {X 0,Y 234.93,Z 530.205,A -85,B 0,C 180,E1 -19650.569,E2 -19650.569} C_VEL
LIN {X 0,Y 234.928,Z 530.207,A -85,B 0,C 180,E1 -19654.639,E2 -19654.639} C_VEL
LIN {X 0,Y 234.94,Z 530.213,A -85,B 0,C 180,E1 -19658.946,E2 -19658.946} C_VEL
LIN {X 0,Y 234.889,Z 530.221,A -85,B 0,C 180,E1 -19663.487,E2 -19663.487} C_VEL
LIN {X 0,Y 234.893,Z 530.322,A -85,B 0,C 180,E1 -19665.043,E2 -19665.043} C_VEL
LIN {X 0,Y 238.637,Z 540.988,A -85,B 0,C 180,E1 -19668.998,E2 -19668.998} C_VEL
LIN {X 0,Y 241.672,Z 551.003,A -85,B 0,C 180,E1 -19672.361,E2 -19672.361} C_VEL
LIN {X 0,Y 242.083,Z 552.135,A -85,B 0,C 180,E1 -19672.603,E2 -19672.603} C_VEL
LIN {X 0,Y 248.182,Z 564.362,A -85,B 0,C 180,E1 -19674.06,E2 -19674.06} C_VEL
LIN {X 0,Y 254.288,Z 578.251,A -85,B 0,C 180,E1 -19675.48,E2 -19675.48} C_VEL
LIN {X 0,Y 256.764,Z 593.443,A -85,B 0,C 180,E1 -19676.342,E2 -19676.342} C_VEL
LIN {X 0,Y 253.882,Z 663.349,A -85,B 0,C 180,E1 -19678.268,E2 -19678.268} C_VEL
LIN {X 0,Y 252.763,Z 676.447,A -85,B 0,C 180,E1 -19678.928,E2 -19678.928} C_VEL
LIN {X 0,Y 251.182,Z 689.444,A -85,B 0,C 180,E1 -19679.93,E2 -19679.93} C_VEL
LIN {X 0,Y 249.418,Z 700.891,A -85,B 0,C 180,E1 -19681.135,E2 -19681.135} C_VEL
LIN {X 0,Y 247.154,Z 712.358,A -85,B 0,C 180,E1 -19682.709,E2 -19682.709} C_VEL
LIN {X 0,Y 244.729,Z 722.596,A -85,B 0,C 180,E1 -19684.485,E2 -19684.485} C_VEL
LIN {X 0,Y 242.3,Z 731.836,A -85,B 0,C 180,E1 -19686.496,E2 -19686.496} C_VEL
LIN {X 0,Y 239.78,Z 740.714,A -85,B 0,C 180,E1 -19688.959,E2 -19688.959} C_VEL
LIN {X 0,Y 237.782,Z 747.86,A -85,B 0,C 180,E1 -19691.475,E2 -19691.475} C_VEL
LIN {X 0,Y 236.454,Z 752.684,A -85,B 0,C 180,E1 -19693.599,E2 -19693.599} C_VEL
LIN {X 0,Y 234.933,Z 757.349,A -85,B 0,C 180,E1 -19696.154,E2 -19696.154} C_VEL
LIN {X 0,Y 234.272,Z 759.849,A -85,B 0,C 180,E1 -19697.878,E2 -19697.878} C_VEL
LIN {X 0,Y 233.73,Z 761.846,A -85,B 0,C 180,E1 -19699.606,E2 -19699.606} C_VEL
LIN {X 0,Y 233.323,Z 763.429,A -85,B 0,C 180,E1 -19701.338,E2 -19701.338} C_VEL
LIN {X 0,Y 233.009,Z 764.616,A -85,B 0,C 180,E1 -19703.071,E2 -19703.071} C_VEL
LIN {X 0,Y 232.776,Z 765.448,A -85,B 0,C 180,E1 -19705.106,E2 -19705.106} C_VEL
LIN {X 0,Y 232.775,Z 765.689,A -85,B 0,C 180,E1 -19708.27,E2 -19708.27} C_VEL
LIN {X 0,Y 232.809,Z 765.28,A -85,B 0,C 180,E1 -19710,E2 -19710} C_VEL
LIN {X 0,Y 233.148,Z 763.2,A -85,B 0,C 180,E1 -19713.456,E2 -19713.456} C_VEL
LIN {X 0,Y 233.63,Z 760.569,A -85,B 0,C 180,E1 -19716.044,E2 -19716.044} C_VEL
LIN {X 0,Y 234.326,Z 756.934,A -85,B 0,C 180,E1 -19718.625,E2 -19718.625} C_VEL
LIN {X 0,Y 235.422,Z 752.185,A -85,B 0,C 180,E1 -19721.189,E2 -19721.189} C_VEL
LIN {X 0,Y 236.874,Z 746.186,A -85,B 0,C 180,E1 -19723.73,E2 -19723.73} C_VEL
LIN {X 0,Y 238.747,Z 738.7,A -85,B 0,C 180,E1 -19726.239,E2 -19726.239} C_VEL
LIN {X 0,Y 240.956,Z 729.285,A -85,B 0,C 180,E1 -19728.713,E2 -19728.713} C_VEL
LIN {X 0,Y 243.114,Z 719.582,A -85,B 0,C 180,E1 -19730.739,E2 -19730.739} C_VEL
LIN {X 0,Y 245.315,Z 708.638,A -85,B 0,C 180,E1 -19732.53,E2 -19732.53} C_VEL
LIN {X 0,Y 247.026,Z 697.982,A -85,B 0,C 180,E1 -19733.917,E2 -19733.917} C_VEL
LIN {X 0,Y 248.716,Z 686.272,A -85,B 0,C 180,E1 -19735.078,E2 -19735.078} C_VEL
LIN {X 0,Y 249.881,Z 674.086,A -85,B 0,C 180,E1 -19735.971,E2 -19735.971} C_VEL
LIN {X 0,Y 250.749,Z 661.146,A -85,B 0,C 180,E1 -19736.588,E2 -19736.588} C_VEL
LIN {X 0,Y 253.392,Z 591.066,A -85,B 0,C 180,E1 -19738.526,E2 -19738.526} C_VEL
LIN {X 0,Y 250.388,Z 572.434,A -85,B 0,C 180,E1 -19739.526,E2 -19739.526} C_VEL
LIN {X 0,Y 244.343,Z 557.901,A -85,B 0,C 180,E1 -19740.863,E2 -19740.863} C_VEL
LIN {X 0,Y 241.306,Z 551.323,A -85,B 0,C 180,E1 -19741.581,E2 -19741.581} C_VEL
LIN {X 0,Y 238.172,Z 540.33,A -85,B 0,C 180,E1 -19745.03,E2 -19745.03} C_VEL
LIN {X 0,Y 235.578,Z 532.266,A -85,B 0,C 180,E1 -19747.761,E2 -19747.761} C_VEL
LIN {X 0,Y 234.978,Z 530.217,A -85,B 0,C 180,E1 -19748.515,E2 -19748.515} C_VEL
LIN {X 0,Y 234.965,Z 530.211,A -85,B 0,C 180,E1 -19753.467,E2 -19753.467} C_VEL
LIN {X 0,Y 234.968,Z 530.198,A -85,B 0,C 180,E1 -19755.754,E2 -19755.754} C_VEL
LIN {X 0,Y 245.394,Z 560.106,A -85,B 0,C 180,E1 -19757.82,E2 -19757.82} C_VEL
LIN {X 0,Y 242.42,Z 627.041,A -85,B 0,C 180,E1 -19760.562,E2 -19760.562} C_VEL
LIN {X 0,Y 241.666,Z 640.899,A -85,B 0,C 180,E1 -19761.464,E2 -19761.464} C_VEL
LIN {X 0,Y 240.594,Z 654.282,A -85,B 0,C 180,E1 -19762.689,E2 -19762.689} C_VEL
LIN {X 0,Y 239.336,Z 667.395,A -85,B 0,C 180,E1 -19764.28,E2 -19764.28} C_VEL
LIN {X 0,Y 238.028,Z 679.222,A -85,B 0,C 180,E1 -19766.13,E2 -19766.13} C_VEL
LIN {X 0,Y 236.759,Z 689.898,A -85,B 0,C 180,E1 -19768.203,E2 -19768.203} C_VEL
LIN {X 0,Y 235.599,Z 699.456,A -85,B 0,C 180,E1 -19770.514,E2 -19770.514} C_VEL
LIN {X 0,Y 234.573,Z 708.696,A -85,B 0,C 180,E1 -19773.293,E2 -19773.293} C_VEL
LIN {X 0,Y 233.973,Z 714.856,A -85,B 0,C 180,E1 -19775.605,E2 -19775.605} C_VEL
LIN {X 0,Y 233.485,Z 719.851,A -85,B 0,C 180,E1 -19777.898,E2 -19777.898} C_VEL
LIN {X 0,Y 233.273,Z 722.804,A -85,B 0,C 180,E1 -19779.543,E2 -19779.543} C_VEL
LIN {X 0,Y 232.475,Z 724.932,A -85,B 0,C 180,E1 -19780.885,E2 -19780.885} C_VEL
LIN {X 0,Y 229.551,Z 727.825,A -85,B 0,C 180,E1 -19783.124,E2 -19783.124} C_VEL
LIN {X 0,Y 227.247,Z 729.732,A -85,B 0,C 180,E1 -19784.985,E2 -19784.985} C_VEL
LIN {X 0,Y 226.393,Z 731.037,A -85,B 0,C 180,E1 -19786.69,E2 -19786.69} C_VEL
LIN {X 0,Y 226.418,Z 731.15,A -85,B 0,C 180,E1 -19786.936,E2 -19786.936} C_VEL
LIN {X 0,Y 227.005,Z 732.279,A -85,B 0,C 180,E1 -19789.294,E2 -19789.294} C_VEL
LIN {X 0,Y 227.687,Z 732.589,A -85,B 0,C 180,E1 -19791.121,E2 -19791.121} C_VEL
LIN {X 0,Y 228.453,Z 732.494,A -85,B 0,C 180,E1 -19792.931,E2 -19792.931} C_VEL
LIN {X 0,Y 229.398,Z 731.986,A -85,B 0,C 180,E1 -19794.726,E2 -19794.726} C_VEL
LIN {X 0,Y 230.54,Z 731,A -85,B 0,C 180,E1 -19796.504,E2 -19796.504} C_VEL
LIN {X 0,Y 232.002,Z 729.413,A -85,B 0,C 180,E1 -19798.458,E2 -19798.458} C_VEL
LIN {X 0,Y 234.129,Z 726.668,A -85,B 0,C 180,E1 -19800.86,E2 -19800.86} C_VEL
LIN {X 0,Y 236.861,Z 722.666,A -85,B 0,C 180,E1 -19803.402,E2 -19803.402} C_VEL
LIN {X 0,Y 240.338,Z 716.831,A -85,B 0,C 180,E1 -19806.168,E2 -19806.168} C_VEL
LIN {X 0,Y 244.177,Z 709.74,A -85,B 0,C 180,E1 -19808.691,E2 -19808.691} C_VEL
LIN {X 0,Y 248.153,Z 701.405,A -85,B 0,C 180,E1 -19811.021,E2 -19811.021} C_VEL
LIN {X 0,Y 251.816,Z 692.841,A -85,B 0,C 180,E1 -19812.901,E2 -19812.901} C_VEL
LIN {X 0,Y 255.743,Z 682.284,A -85,B 0,C 180,E1 -19814.754,E2 -19814.754} C_VEL
LIN {X 0,Y 259.415,Z 670.91,A -85,B 0,C 180,E1 -19816.324,E2 -19816.324} C_VEL
LIN {X 0,Y 262.763,Z 657.862,A -85,B 0,C 180,E1 -19817.712,E2 -19817.712} C_VEL
LIN {X 0,Y 265.391,Z 644.562,A -85,B 0,C 180,E1 -19818.779,E2 -19818.779} C_VEL
LIN {X 0,Y 267.178,Z 632.932,A -85,B 0,C 180,E1 -19819.446,E2 -19819.446} C_VEL
LIN {X 0,Y 270.979,Z 602.78,A -85,B 0,C 180,E1 -19820.726,E2 -19820.726} C_VEL
LIN {X 0,Y 272.548,Z 590.484,A -85,B 0,C 180,E1 -19821.245,E2 -19821.245} C_VEL
LIN {X 0,Y 269.661,Z 585.165,A -85,B 0,C 180,E1 -19822.959,E2 -19822.959} C_VEL
LIN {X 0,Y 267.055,Z 580.803,A -85,B 0,C 180,E1 -19824.708,E2 -19824.708} C_VEL
LIN {X 0,Y 263.99,Z 576.38,A -85,B 0,C 180,E1 -19827.161,E2 -19827.161} C_VEL
LIN {X 0,Y 261.684,Z 573.402,A -85,B 0,C 180,E1 -19829.57,E2 -19829.57} C_VEL
LIN {X 0,Y 259.161,Z 571.178,A -85,B 0,C 180,E1 -19833.869,E2 -19833.869} C_VEL
LIN {X 0,Y 258.665,Z 571.741,A -85,B 0,C 180,E1 -19836.709,E2 -19836.709} C_VEL
LIN {X 0,Y 259.149,Z 573.479,A -85,B 0,C 180,E1 -19839.6,E2 -19839.6} C_VEL
LIN {X 0,Y 259.619,Z 575.055,A -85,B 0,C 180,E1 -19840.956,E2 -19840.956} C_VEL
LIN {X 0,Y 262.406,Z 581.431,A -85,B 0,C 180,E1 -19844.965,E2 -19844.965} C_VEL
LIN {X 0,Y 265.173,Z 588.372,A -85,B 0,C 180,E1 -19847.665,E2 -19847.665} C_VEL
LIN {X 0,Y 267.243,Z 594.009,A -85,B 0,C 180,E1 -19849.346,E2 -19849.346} C_VEL
LIN {X 0,Y 269.444,Z 600.442,A -85,B 0,C 180,E1 -19850.95,E2 -19850.95} C_VEL
LIN {X 0,Y 269.72,Z 605.891,A -85,B 0,C 180,E1 -19851.554,E2 -19851.554} C_VEL
LIN {X 0,Y 269.772,Z 616.704,A -85,B 0,C 180,E1 -19852.517,E2 -19852.517} C_VEL
LIN {X 0,Y 269.441,Z 621.553,A -85,B 0,C 180,E1 -19852.815,E2 -19852.815} C_VEL
LIN {X 0,Y 264.663,Z 658.544,A -85,B 0,C 180,E1 -19854.372,E2 -19854.372} C_VEL
LIN {X 0,Y 262.013,Z 671.906,A -85,B 0,C 180,E1 -19855.134,E2 -19855.134} C_VEL
LIN {X 0,Y 258.624,Z 684.924,A -85,B 0,C 180,E1 -19856.147,E2 -19856.147} C_VEL
LIN {X 0,Y 254.696,Z 697.517,A -85,B 0,C 180,E1 -19857.448,E2 -19857.448} C_VEL
LIN {X 0,Y 250.14,Z 710.059,A -85,B 0,C 180,E1 -19859.153,E2 -19859.153} C_VEL
LIN {X 0,Y 246.051,Z 720.352,A -85,B 0,C 180,E1 -19860.951,E2 -19860.951} C_VEL
LIN {X 0,Y 241.614,Z 730.418,A -85,B 0,C 180,E1 -19863.202,E2 -19863.202} C_VEL
LIN {X 0,Y 237.677,Z 738.748,A -85,B 0,C 180,E1 -19865.546,E2 -19865.546} C_VEL
LIN {X 0,Y 234.386,Z 745.614,A -85,B 0,C 180,E1 -19867.988,E2 -19867.988} C_VEL
LIN {X 0,Y 231.709,Z 751.193,A -85,B 0,C 180,E1 -19870.51,E2 -19870.51} C_VEL
LIN {X 0,Y 229.667,Z 755.578,A -85,B 0,C 180,E1 -19872.871,E2 -19872.871} C_VEL
LIN {X 0,Y 227.882,Z 762.739,A -85,B 0,C 180,E1 -19875.717,E2 -19875.717} C_VEL
LIN {X 0,Y 226.782,Z 767.938,A -85,B 0,C 180,E1 -19878.379,E2 -19878.379} C_VEL
LIN {X 0,Y 226.125,Z 771.955,A -85,B 0,C 180,E1 -19881.06,E2 -19881.06} C_VEL
LIN {X 0,Y 225.848,Z 774.017,A -85,B 0,C 180,E1 -19882.85,E2 -19882.85} C_VEL
LIN {X 0,Y 225.67,Z 776.136,A -85,B 0,C 180,E1 -19885.252,E2 -19885.252} C_VEL
LIN {X 0,Y 225.692,Z 777.673,A -85,B 0,C 180,E1 -19888.216,E2 -19888.216} C_VEL
LIN {X 0,Y 225.723,Z 778.045,A -85,B 0,C 180,E1 -19890,E2 -19890} C_VEL
LIN {X 0,Y 225.688,Z 778.026,A -85,B 0,C 180,E1 -19891.784,E2 -19891.784} C_VEL
LIN {X 0,Y 225.676,Z 777.087,A -85,B 0,C 180,E1 -19894.767,E2 -19894.767} C_VEL
LIN {X 0,Y 225.842,Z 775.502,A -85,B 0,C 180,E1 -19897.15,E2 -19897.15} C_VEL
LIN {X 0,Y 226.358,Z 772.828,A -85,B 0,C 180,E1 -19899.832,E2 -19899.832} C_VEL
LIN {X 0,Y 227.21,Z 769.13,A -85,B 0,C 180,E1 -19902.505,E2 -19902.505} C_VEL
LIN {X 0,Y 228.524,Z 764.305,A -85,B 0,C 180,E1 -19905.153,E2 -19905.153} C_VEL
LIN {X 0,Y 230.346,Z 758.208,A -85,B 0,C 180,E1 -19907.764,E2 -19907.764} C_VEL
LIN {X 0,Y 232.451,Z 751.008,A -85,B 0,C 180,E1 -19910.217,E2 -19910.217} C_VEL
LIN {X 0,Y 234.654,Z 742.831,A -85,B 0,C 180,E1 -19912.449,E2 -19912.449} C_VEL
LIN {X 0,Y 237.185,Z 733.317,A -85,B 0,C 180,E1 -19914.508,E2 -19914.508} C_VEL
LIN {X 0,Y 239.827,Z 722.759,A -85,B 0,C 180,E1 -19916.309,E2 -19916.309} C_VEL
LIN {X 0,Y 241.985,Z 712.54,A -85,B 0,C 180,E1 -19917.689,E2 -19917.689} C_VEL
LIN {X 0,Y 244.11,Z 700.294,A -85,B 0,C 180,E1 -19918.949,E2 -19918.949} C_VEL
LIN {X 0,Y 245.924,Z 687.461,A -85,B 0,C 180,E1 -19919.889,E2 -19919.889} C_VEL
LIN {X 0,Y 247.08,Z 674.841,A -85,B 0,C 180,E1 -19920.5,E2 -19920.5} C_VEL
LIN {X 0,Y 249.447,Z 614.966,A -85,B 0,C 180,E1 -19922.2,E2 -19922.2} C_VEL
LIN {X 0,Y 246.265,Z 585.622,A -85,B 0,C 180,E1 -19923.692,E2 -19923.692} C_VEL
LIN {X 0,Y 244.329,Z 572.9,A -85,B 0,C 180,E1 -19924.452,E2 -19924.452} C_VEL
LIN {X 0,Y 238.542,Z 557.977,A -85,B 0,C 180,E1 -19926.046,E2 -19926.046} C_VEL
LIN {X 0,Y 235.694,Z 547.3,A -85,B 0,C 180,E1 -19928.145,E2 -19928.145} C_VEL
LIN {X 0,Y 229.588,Z 534.923,A -85,B 0,C 180,E1 -19931.347,E2 -19931.347} C_VEL
LIN {X 0,Y 228.405,Z 533.115,A -85,B 0,C 180,E1 -19931.939,E2 -19931.939} C_VEL
LIN {X 0,Y 227.838,Z 531.1,A -85,B 0,C 180,E1 -19932.494,E2 -19932.494} C_VEL
LIN {X 0,Y 227.892,Z 531.087,A -85,B 0,C 180,E1 -19937.277,E2 -19937.277} C_VEL
LIN {X 0,Y 227.868,Z 531.092,A -85,B 0,C 180,E1 -19941.914,E2 -19941.914} C_VEL
LIN {X 0,Y 227.887,Z 531.099,A -85,B 0,C 180,E1 -19946.372,E2 -19946.372} C_VEL
LIN {X 0,Y 227.915,Z 531.076,A -85,B 0,C 180,E1 -19950.437,E2 -19950.437} C_VEL
LIN {X 0,Y 227.92,Z 531.074,A -85,B 0,C 180,E1 -19954.425,E2 -19954.425} C_VEL
LIN {X 0,Y 227.943,Z 531.081,A -85,B 0,C 180,E1 -19958.285,E2 -19958.285} C_VEL
LIN {X 0,Y 228.029,Z 531.049,A -85,B 0,C 180,E1 -19962.827,E2 -19962.827} C_VEL
LIN {X 0,Y 228.087,Z 531.074,A -85,B 0,C 180,E1 -19967.544,E2 -19967.544} C_VEL
LIN {X 0,Y 228.3,Z 531.012,A -85,B 0,C 180,E1 -19971.146,E2 -19971.146} C_VEL
LIN {X 0,Y 228.349,Z 531.011,A -85,B 0,C 180,E1 -19972.929,E2 -19972.929} C_VEL
LIN {X 0,Y 228.55,Z 530.992,A -85,B 0,C 180,E1 -19978.238,E2 -19978.238} C_VEL
LIN {X 0,Y 228.55,Z 530.99,A -85,B 0,C 180,E1 -19981.763,E2 -19981.763} C_VEL
LIN {X 0,Y 228.32,Z 531.016,A -85,B 0,C 180,E1 -19987.073,E2 -19987.073} C_VEL
LIN {X 0,Y 228.141,Z 531.053,A -85,B 0,C 180,E1 -19990.652,E2 -19990.652} C_VEL
LIN {X 0,Y 228.055,Z 531.061,A -85,B 0,C 180,E1 -19994.273,E2 -19994.273} C_VEL
LIN {X 0,Y 227.999,Z 531.065,A -85,B 0,C 180,E1 -19997.954,E2 -19997.954} C_VEL
LIN {X 0,Y 227.926,Z 531.072,A -85,B 0,C 180,E1 -20002.33,E2 -20002.33} C_VEL
LIN {X 0,Y 227.941,Z 531.093,A -85,B 0,C 180,E1 -20006.604,E2 -20006.604} C_VEL
LIN {X 0,Y 227.907,Z 531.077,A -85,B 0,C 180,E1 -20010.297,E2 -20010.297} C_VEL
LIN {X 0,Y 227.875,Z 531.091,A -85,B 0,C 180,E1 -20013.721,E2 -20013.721} C_VEL
LIN {X 0,Y 227.842,Z 531.104,A -85,B 0,C 180,E1 -20018.092,E2 -20018.092} C_VEL
LIN {X 0,Y 227.811,Z 531.105,A -85,B 0,C 180,E1 -20022.743,E2 -20022.743} C_VEL
LIN {X 0,Y 227.855,Z 531.194,A -85,B 0,C 180,E1 -20023.642,E2 -20023.642} C_VEL
LIN {X 0,Y 231.662,Z 541.854,A -85,B 0,C 180,E1 -20027.793,E2 -20027.793} C_VEL
LIN {X 0,Y 234.96,Z 552.053,A -85,B 0,C 180,E1 -20031.308,E2 -20031.308} C_VEL
LIN {X 0,Y 242.311,Z 566.564,A -85,B 0,C 180,E1 -20033.163,E2 -20033.163} C_VEL
LIN {X 0,Y 248.639,Z 581.008,A -85,B 0,C 180,E1 -20034.707,E2 -20034.707} C_VEL
LIN {X 0,Y 250.805,Z 594.305,A -85,B 0,C 180,E1 -20035.494,E2 -20035.494} C_VEL
LIN {X 0,Y 247.883,Z 662.671,A -85,B 0,C 180,E1 -20037.406,E2 -20037.406} C_VEL
LIN {X 0,Y 246.784,Z 675.425,A -85,B 0,C 180,E1 -20038.028,E2 -20038.028} C_VEL
LIN {X 0,Y 245.303,Z 687.701,A -85,B 0,C 180,E1 -20038.956,E2 -20038.956} C_VEL
LIN {X 0,Y 243.321,Z 700.011,A -85,B 0,C 180,E1 -20040.228,E2 -20040.228} C_VEL
LIN {X 0,Y 241.161,Z 711.094,A -85,B 0,C 180,E1 -20041.735,E2 -20041.735} C_VEL
LIN {X 0,Y 238.61,Z 721.58,A -85,B 0,C 180,E1 -20043.546,E2 -20043.546} C_VEL
LIN {X 0,Y 235.775,Z 731.898,A -85,B 0,C 180,E1 -20045.805,E2 -20045.805} C_VEL
LIN {X 0,Y 233.14,Z 740.803,A -85,B 0,C 180,E1 -20048.33,E2 -20048.33} C_VEL
LIN {X 0,Y 231.029,Z 747.967,A -85,B 0,C 180,E1 -20050.913,E2 -20050.913} C_VEL
LIN {X 0,Y 229.626,Z 752.807,A -85,B 0,C 180,E1 -20053.097,E2 -20053.097} C_VEL
LIN {X 0,Y 228.012,Z 757.488,A -85,B 0,C 180,E1 -20055.725,E2 -20055.725} C_VEL
LIN {X 0,Y 226.991,Z 761.046,A -85,B 0,C 180,E1 -20058.39,E2 -20058.39} C_VEL
LIN {X 0,Y 226.283,Z 763.594,A -85,B 0,C 180,E1 -20061.066,E2 -20061.066} C_VEL
LIN {X 0,Y 225.943,Z 764.787,A -85,B 0,C 180,E1 -20062.853,E2 -20062.853} C_VEL
LIN {X 0,Y 225.688,Z 765.697,A -85,B 0,C 180,E1 -20065.206,E2 -20065.206} C_VEL
LIN {X 0,Y 225.69,Z 765.883,A -85,B 0,C 180,E1 -20068.216,E2 -20068.216} C_VEL
LIN {X 0,Y 225.722,Z 765.481,A -85,B 0,C 180,E1 -20070,E2 -20070} C_VEL
LIN {X 0,Y 226.076,Z 763.417,A -85,B 0,C 180,E1 -20073.565,E2 -20073.565} C_VEL
LIN {X 0,Y 226.634,Z 760.377,A -85,B 0,C 180,E1 -20076.594,E2 -20076.594} C_VEL
LIN {X 0,Y 227.659,Z 755.743,A -85,B 0,C 180,E1 -20079.775,E2 -20079.775} C_VEL
LIN {X 0,Y 228.948,Z 750.599,A -85,B 0,C 180,E1 -20082.408,E2 -20082.408} C_VEL
LIN {X 0,Y 230.619,Z 744.133,A -85,B 0,C 180,E1 -20085.012,E2 -20085.012} C_VEL
LIN {X 0,Y 232.679,Z 736.095,A -85,B 0,C 180,E1 -20087.58,E2 -20087.58} C_VEL
LIN {X 0,Y 234.721,Z 727.847,A -85,B 0,C 180,E1 -20089.684,E2 -20089.684} C_VEL
LIN {X 0,Y 236.942,Z 717.679,A -85,B 0,C 180,E1 -20091.762,E2 -20091.762} C_VEL
LIN {X 0,Y 239.391,Z 706.261,A -85,B 0,C 180,E1 -20093.578,E2 -20093.578} C_VEL
LIN {X 0,Y 241.199,Z 694.863,A -85,B 0,C 180,E1 -20094.992,E2 -20094.992} C_VEL
LIN {X 0,Y 242.787,Z 682.501,A -85,B 0,C 180,E1 -20096.144,E2 -20096.144} C_VEL
LIN {X 0,Y 243.974,Z 669.84,A -85,B 0,C 180,E1 -20096.98,E2 -20096.98} C_VEL
LIN {X 0,Y 244.749,Z 656.186,A -85,B 0,C 180,E1 -20097.523,E2 -20097.523} C_VEL
LIN {X 0,Y 247.172,Z 591.421,A -85,B 0,C 180,E1 -20099.338,E2 -20099.338} C_VEL
LIN {X 0,Y 244.41,Z 574.768,A -85,B 0,C 180,E1 -20100.281,E2 -20100.281} C_VEL
LIN {X 0,Y 239.084,Z 561.777,A -85,B 0,C 180,E1 -20101.517,E2 -20101.517} C_VEL
LIN {X 0,Y 234.196,Z 551.492,A -85,B 0,C 180,E1 -20102.694,E2 -20102.694} C_VEL
LIN {X 0,Y 230.707,Z 539.538,A -85,B 0,C 180,E1 -20106.621,E2 -20106.621} C_VEL
LIN {X 0,Y 227.887,Z 531.087,A -85,B 0,C 180,E1 -20109.707,E2 -20109.707} C_VEL
LIN {X 0,Y 227.909,Z 531.099,A -85,B 0,C 180,E1 -20112.718,E2 -20112.718} C_VEL
LIN {X 0,Y 227.89,Z 531.078,A -85,B 0,C 180,E1 -20115.256,E2 -20115.256} C_VEL
LIN {X 0,Y 238.475,Z 561.987,A -85,B 0,C 180,E1 -20117.455,E2 -20117.455} C_VEL
LIN {X 0,Y 235.409,Z 627.898,A -85,B 0,C 180,E1 -20120.277,E2 -20120.277} C_VEL
LIN {X 0,Y 234.607,Z 642.413,A -85,B 0,C 180,E1 -20121.266,E2 -20121.266} C_VEL
LIN {X 0,Y 233.436,Z 655.901,A -85,B 0,C 180,E1 -20122.57,E2 -20122.57} C_VEL
LIN {X 0,Y 232.252,Z 668.054,A -85,B 0,C 180,E1 -20124.105,E2 -20124.105} C_VEL
LIN {X 0,Y 230.937,Z 679.803,A -85,B 0,C 180,E1 -20125.999,E2 -20125.999} C_VEL
LIN {X 0,Y 229.637,Z 690.481,A -85,B 0,C 180,E1 -20128.133,E2 -20128.133} C_VEL
LIN {X 0,Y 228.473,Z 700.052,A -85,B 0,C 180,E1 -20130.516,E2 -20130.516} C_VEL
LIN {X 0,Y 227.527,Z 708.593,A -85,B 0,C 180,E1 -20133.141,E2 -20133.141} C_VEL
LIN {X 0,Y 226.839,Z 715.434,A -85,B 0,C 180,E1 -20135.762,E2 -20135.762} C_VEL
LIN {X 0,Y 226.283,Z 721.467,A -85,B 0,C 180,E1 -20138.706,E2 -20138.706} C_VEL
LIN {X 0,Y 226.013,Z 726.386,A -85,B 0,C 180,E1 -20141.883,E2 -20141.883} C_VEL
LIN {X 0,Y 226.099,Z 729.296,A -85,B 0,C 180,E1 -20144.487,E2 -20144.487} C_VEL
LIN {X 0,Y 226.418,Z 731.15,A -85,B 0,C 180,E1 -20146.936,E2 -20146.936} C_VEL
LIN {X 0,Y 226.091,Z 732.052,A -85,B 0,C 180,E1 -20148.414,E2 -20148.414} C_VEL
LIN {X 0,Y 224.008,Z 733.044,A -85,B 0,C 180,E1 -20150.872,E2 -20150.872} C_VEL
LIN {X 0,Y 222.232,Z 733.219,A -85,B 0,C 180,E1 -20153.383,E2 -20153.383} C_VEL
LIN {X 0,Y 222.391,Z 732.84,A -85,B 0,C 180,E1 -20154.905,E2 -20154.905} C_VEL
LIN {X 0,Y 224.688,Z 731.134,A -85,B 0,C 180,E1 -20158.207,E2 -20158.207} C_VEL
LIN {X 0,Y 226.993,Z 728.607,A -85,B 0,C 180,E1 -20160.887,E2 -20160.887} C_VEL
LIN {X 0,Y 229.793,Z 725.013,A -85,B 0,C 180,E1 -20163.506,E2 -20163.506} C_VEL
LIN {X 0,Y 233.326,Z 719.836,A -85,B 0,C 180,E1 -20166.297,E2 -20166.297} C_VEL
LIN {X 0,Y 237.33,Z 713.236,A -85,B 0,C 180,E1 -20168.944,E2 -20168.944} C_VEL
LIN {X 0,Y 241.462,Z 705.524,A -85,B 0,C 180,E1 -20171.33,E2 -20171.33} C_VEL
LIN {X 0,Y 245.789,Z 696.428,A -85,B 0,C 180,E1 -20173.552,E2 -20173.552} C_VEL
LIN {X 0,Y 250.054,Z 686.232,A -85,B 0,C 180,E1 -20175.486,E2 -20175.486} C_VEL
LIN {X 0,Y 253.919,Z 675.368,A -85,B 0,C 180,E1 -20177.102,E2 -20177.102} C_VEL
LIN {X 0,Y 257.445,Z 663.556,A -85,B 0,C 180,E1 -20178.503,E2 -20178.503} C_VEL
LIN {X 0,Y 260.391,Z 651.352,A -85,B 0,C 180,E1 -20179.614,E2 -20179.614} C_VEL
LIN {X 0,Y 262.865,Z 637.385,A -85,B 0,C 180,E1 -20180.559,E2 -20180.559} C_VEL
LIN {X 0,Y 266.839,Z 607.853,A -85,B 0,C 180,E1 -20181.851,E2 -20181.851} C_VEL
LIN {X 0,Y 268.678,Z 594.367,A -85,B 0,C 180,E1 -20182.443,E2 -20182.443} C_VEL
LIN {X 0,Y 265.651,Z 588.665,A -85,B 0,C 180,E1 -20184.487,E2 -20184.487} C_VEL
LIN {X 0,Y 263.118,Z 584.816,A -85,B 0,C 180,E1 -20186.434,E2 -20186.434} C_VEL
LIN {X 0,Y 261.842,Z 582.851,A -85,B 0,C 180,E1 -20187.66,E2 -20187.66} C_VEL
LIN {X 0,Y 259.957,Z 580.222,A -85,B 0,C 180,E1 -20189.786,E2 -20189.786} C_VEL
LIN {X 0,Y 257.798,Z 578.281,A -85,B 0,C 180,E1 -20193.44,E2 -20193.44} C_VEL
LIN {X 0,Y 257.273,Z 578.299,A -85,B 0,C 180,E1 -20195.511,E2 -20195.511} C_VEL
LIN {X 0,Y 257.331,Z 579.855,A -85,B 0,C 180,E1 -20198.74,E2 -20198.74} C_VEL
LIN {X 0,Y 257.857,Z 581.414,A -85,B 0,C 180,E1 -20200.379,E2 -20200.379} C_VEL
LIN {X 0,Y 260.22,Z 587.694,A -85,B 0,C 180,E1 -20204.388,E2 -20204.388} C_VEL
LIN {X 0,Y 262.714,Z 594.543,A -85,B 0,C 180,E1 -20207.086,E2 -20207.086} C_VEL
LIN {X 0,Y 264.355,Z 599.474,A -85,B 0,C 180,E1 -20208.591,E2 -20208.591} C_VEL
LIN {X 0,Y 266.121,Z 604.908,A -85,B 0,C 180,E1 -20209.984,E2 -20209.984} C_VEL
LIN {X 0,Y 266.032,Z 616.898,A -85,B 0,C 180,E1 -20211.156,E2 -20211.156} C_VEL
LIN {X 0,Y 265.813,Z 621.611,A -85,B 0,C 180,E1 -20211.509,E2 -20211.509} C_VEL
LIN {X 0,Y 260.941,Z 657.268,A -85,B 0,C 180,E1 -20213.004,E2 -20213.004} C_VEL
LIN {X 0,Y 258.032,Z 671.11,A -85,B 0,C 180,E1 -20213.794,E2 -20213.794} C_VEL
LIN {X 0,Y 254.518,Z 683.93,A -85,B 0,C 180,E1 -20214.802,E2 -20214.802} C_VEL
LIN {X 0,Y 250.401,Z 696.598,A -85,B 0,C 180,E1 -20216.095,E2 -20216.095} C_VEL
LIN {X 0,Y 245.608,Z 709.122,A -85,B 0,C 180,E1 -20217.796,E2 -20217.796} C_VEL
LIN {X 0,Y 241.609,Z 718.403,A -85,B 0,C 180,E1 -20219.401,E2 -20219.401} C_VEL
LIN {X 0,Y 236.854,Z 728.689,A -85,B 0,C 180,E1 -20221.657,E2 -20221.657} C_VEL
LIN {X 0,Y 232.57,Z 737.154,A -85,B 0,C 180,E1 -20224.013,E2 -20224.013} C_VEL
LIN {X 0,Y 228.382,Z 745.149,A -85,B 0,C 180,E1 -20226.899,E2 -20226.899} C_VEL
LIN {X 0,Y 225.037,Z 751.479,A -85,B 0,C 180,E1 -20229.908,E2 -20229.908} C_VEL
LIN {X 0,Y 222.7,Z 755.926,A -85,B 0,C 180,E1 -20232.555,E2 -20232.555} C_VEL
LIN {X 0,Y 220.989,Z 762.486,A -85,B 0,C 180,E1 -20235.261,E2 -20235.261} C_VEL
LIN {X 0,Y 219.791,Z 767.698,A -85,B 0,C 180,E1 -20238.004,E2 -20238.004} C_VEL
LIN {X 0,Y 219.071,Z 771.727,A -85,B 0,C 180,E1 -20240.77,E2 -20240.77} C_VEL
LIN {X 0,Y 218.799,Z 773.798,A -85,B 0,C 180,E1 -20242.618,E2 -20242.618} C_VEL
LIN {X 0,Y 218.575,Z 776.108,A -85,B 0,C 180,E1 -20245.39,E2 -20245.39} C_VEL
LIN {X 0,Y 218.588,Z 777.474,A -85,B 0,C 180,E1 -20248.158,E2 -20248.158} C_VEL
LIN {X 0,Y 218.639,Z 777.852,A -85,B 0,C 180,E1 -20250,E2 -20250} C_VEL
LIN {X 0,Y 218.585,Z 777.837,A -85,B 0,C 180,E1 -20251.842,E2 -20251.842} C_VEL
LIN {X 0,Y 218.566,Z 777.057,A -85,B 0,C 180,E1 -20254.582,E2 -20254.582} C_VEL
LIN {X 0,Y 218.793,Z 775.334,A -85,B 0,C 180,E1 -20257.382,E2 -20257.382} C_VEL
LIN {X 0,Y 219.339,Z 772.67,A -85,B 0,C 180,E1 -20260.15,E2 -20260.15} C_VEL
LIN {X 0,Y 220.23,Z 768.984,A -85,B 0,C 180,E1 -20262.908,E2 -20262.908} C_VEL
LIN {X 0,Y 221.663,Z 764.172,A -85,B 0,C 180,E1 -20265.634,E2 -20265.634} C_VEL
LIN {X 0,Y 223.549,Z 758.089,A -85,B 0,C 180,E1 -20268.323,E2 -20268.323} C_VEL
LIN {X 0,Y 225.595,Z 751.5,A -85,B 0,C 180,E1 -20270.649,E2 -20270.649} C_VEL
LIN {X 0,Y 228.076,Z 742.758,A -85,B 0,C 180,E1 -20273.133,E2 -20273.133} C_VEL
LIN {X 0,Y 230.757,Z 733.269,A -85,B 0,C 180,E1 -20275.238,E2 -20275.238} C_VEL
LIN {X 0,Y 233.485,Z 722.742,A -85,B 0,C 180,E1 -20277.081,E2 -20277.081} C_VEL
LIN {X 0,Y 235.73,Z 712.569,A -85,B 0,C 180,E1 -20278.49,E2 -20278.49} C_VEL
LIN {X 0,Y 237.945,Z 700.411,A -85,B 0,C 180,E1 -20279.773,E2 -20279.773} C_VEL
LIN {X 0,Y 239.789,Z 687.688,A -85,B 0,C 180,E1 -20280.735,E2 -20280.735} C_VEL
LIN {X 0,Y 241.023,Z 675.421,A -85,B 0,C 180,E1 -20281.352,E2 -20281.352} C_VEL
LIN {X 0,Y 243.477,Z 615.564,A -85,B 0,C 180,E1 -20283.098,E2 -20283.098} C_VEL
LIN {X 0,Y 240.386,Z 586.47,A -85,B 0,C 180,E1 -20284.632,E2 -20284.632} C_VEL
LIN {X 0,Y 238.789,Z 575.576,A -85,B 0,C 180,E1 -20285.301,E2 -20285.301} C_VEL
LIN {X 0,Y 232.039,Z 558.591,A -85,B 0,C 180,E1 -20287.178,E2 -20287.178} C_VEL
LIN {X 0,Y 229.858,Z 550.52,A -85,B 0,C 180,E1 -20288.835,E2 -20288.835} C_VEL
LIN {X 0,Y 224.466,Z 539.565,A -85,B 0,C 180,E1 -20291.804,E2 -20291.804} C_VEL
LIN {X 0,Y 221.003,Z 533.137,A -85,B 0,C 180,E1 -20293.834,E2 -20293.834} C_VEL
LIN {X 0,Y 220.779,Z 531.973,A -85,B 0,C 180,E1 -20294.188,E2 -20294.188} C_VEL
LIN {X 0,Y 220.83,Z 531.962,A -85,B 0,C 180,E1 -20298.062,E2 -20298.062} C_VEL
LIN {X 0,Y 220.831,Z 531.959,A -85,B 0,C 180,E1 -20302.794,E2 -20302.794} C_VEL
LIN {X 0,Y 220.821,Z 531.972,A -85,B 0,C 180,E1 -20307.245,E2 -20307.245} C_VEL
LIN {X 0,Y 220.832,Z 531.97,A -85,B 0,C 180,E1 -20311.486,E2 -20311.486} C_VEL
LIN {X 0,Y 220.857,Z 531.943,A -85,B 0,C 180,E1 -20315.564,E2 -20315.564} C_VEL
LIN {X 0,Y 220.879,Z 531.971,A -85,B 0,C 180,E1 -20319.513,E2 -20319.513} C_VEL
LIN {X 0,Y 221.009,Z 531.92,A -85,B 0,C 180,E1 -20323.37,E2 -20323.37} C_VEL
LIN {X 0,Y 221.107,Z 531.933,A -85,B 0,C 180,E1 -20329.006,E2 -20329.006} C_VEL
LIN {X 0,Y 221.284,Z 531.888,A -85,B 0,C 180,E1 -20332.702,E2 -20332.702} C_VEL
LIN {X 0,Y 221.508,Z 531.869,A -85,B 0,C 180,E1 -20338.182,E2 -20338.182} C_VEL
LIN {X 0,Y 221.508,Z 531.867,A -85,B 0,C 180,E1 -20341.819,E2 -20341.819} C_VEL
LIN {X 0,Y 221.255,Z 531.893,A -85,B 0,C 180,E1 -20347.3,E2 -20347.3} C_VEL
LIN {X 0,Y 221.063,Z 531.94,A -85,B 0,C 180,E1 -20350.997,E2 -20350.997} C_VEL
LIN {X 0,Y 221.01,Z 531.923,A -85,B 0,C 180,E1 -20356.631,E2 -20356.631} C_VEL
LIN {X 0,Y 220.889,Z 531.97,A -85,B 0,C 180,E1 -20360.487,E2 -20360.487} C_VEL
LIN {X 0,Y 220.864,Z 531.952,A -85,B 0,C 180,E1 -20364.436,E2 -20364.436} C_VEL
LIN {X 0,Y 220.835,Z 531.96,A -85,B 0,C 180,E1 -20368.514,E2 -20368.514} C_VEL
LIN {X 0,Y 220.816,Z 531.98,A -85,B 0,C 180,E1 -20372.757,E2 -20372.757} C_VEL
LIN {X 0,Y 220.809,Z 531.986,A -85,B 0,C 180,E1 -20377.28,E2 -20377.28} C_VEL
LIN {X 0,Y 220.77,Z 531.991,A -85,B 0,C 180,E1 -20381.953,E2 -20381.953} C_VEL
LIN {X 0,Y 220.898,Z 532.726,A -85,B 0,C 180,E1 -20382.339,E2 -20382.339} C_VEL
LIN {X 0,Y 224.348,Z 541.746,A -85,B 0,C 180,E1 -20386.097,E2 -20386.097} C_VEL
LIN {X 0,Y 227.384,Z 550.943,A -85,B 0,C 180,E1 -20389.53,E2 -20389.53} C_VEL
LIN {X 0,Y 227.851,Z 552.283,A -85,B 0,C 180,E1 -20389.921,E2 -20389.921} C_VEL
LIN {X 0,Y 234.501,Z 564.644,A -85,B 0,C 180,E1 -20391.698,E2 -20391.698} C_VEL
LIN {X 0,Y 241.879,Z 580.958,A -85,B 0,C 180,E1 -20393.605,E2 -20393.605} C_VEL
LIN {X 0,Y 243.287,Z 585.048,A -85,B 0,C 180,E1 -20393.985,E2 -20393.985} C_VEL
LIN {X 0,Y 244.876,Z 595.447,A -85,B 0,C 180,E1 -20394.61,E2 -20394.61} C_VEL
LIN {X 0,Y 241.82,Z 663.32,A -85,B 0,C 180,E1 -20396.546,E2 -20396.546} C_VEL
LIN {X 0,Y 240.631,Z 676.618,A -85,B 0,C 180,E1 -20397.233,E2 -20397.233} C_VEL
LIN {X 0,Y 238.924,Z 689.45,A -85,B 0,C 180,E1 -20398.25,E2 -20398.25} C_VEL
LIN {X 0,Y 237.004,Z 700.926,A -85,B 0,C 180,E1 -20399.494,E2 -20399.494} C_VEL
LIN {X 0,Y 234.624,Z 712.343,A -85,B 0,C 180,E1 -20401.118,E2 -20401.118} C_VEL
LIN {X 0,Y 231.954,Z 722.651,A -85,B 0,C 180,E1 -20402.969,E2 -20402.969} C_VEL
LIN {X 0,Y 229.291,Z 731.958,A -85,B 0,C 180,E1 -20405.074,E2 -20405.074} C_VEL
LIN {X 0,Y 226.519,Z 740.892,A -85,B 0,C 180,E1 -20407.663,E2 -20407.663} C_VEL
LIN {X 0,Y 224.381,Z 747.809,A -85,B 0,C 180,E1 -20410.209,E2 -20410.209} C_VEL
LIN {X 0,Y 222.812,Z 752.931,A -85,B 0,C 180,E1 -20412.564,E2 -20412.564} C_VEL
LIN {X 0,Y 221.107,Z 757.626,A -85,B 0,C 180,E1 -20415.269,E2 -20415.269} C_VEL
LIN {X 0,Y 220.026,Z 761.198,A -85,B 0,C 180,E1 -20418.017,E2 -20418.017} C_VEL
LIN {X 0,Y 219.264,Z 763.758,A -85,B 0,C 180,E1 -20420.778,E2 -20420.778} C_VEL
LIN {X 0,Y 218.903,Z 764.957,A -85,B 0,C 180,E1 -20422.622,E2 -20422.622} C_VEL
LIN {X 0,Y 218.586,Z 765.958,A -85,B 0,C 180,E1 -20425.364,E2 -20425.364} C_VEL
LIN {X 0,Y 218.588,Z 766.077,A -85,B 0,C 180,E1 -20428.158,E2 -20428.158} C_VEL
LIN {X 0,Y 218.638,Z 765.682,A -85,B 0,C 180,E1 -20430,E2 -20430} C_VEL
LIN {X 0,Y 218.737,Z 764.859,A -85,B 0,C 180,E1 -20431.841,E2 -20431.841} C_VEL
LIN {X 0,Y 219.007,Z 763.633,A -85,B 0,C 180,E1 -20433.68,E2 -20433.68} C_VEL
LIN {X 0,Y 219.509,Z 760.975,A -85,B 0,C 180,E1 -20436.481,E2 -20436.481} C_VEL
LIN {X 0,Y 220.296,Z 757.418,A -85,B 0,C 180,E1 -20439.178,E2 -20439.178} C_VEL
LIN {X 0,Y 221.52,Z 752.696,A -85,B 0,C 180,E1 -20441.901,E2 -20441.901} C_VEL
LIN {X 0,Y 223.15,Z 746.724,A -85,B 0,C 180,E1 -20444.593,E2 -20444.593} C_VEL
LIN {X 0,Y 225.2,Z 739.282,A -85,B 0,C 180,E1 -20447.246,E2 -20447.246} C_VEL
LIN {X 0,Y 227.564,Z 729.913,A -85,B 0,C 180,E1 -20449.859,E2 -20449.859} C_VEL
LIN {X 0,Y 229.93,Z 720.259,A -85,B 0,C 180,E1 -20451.989,E2 -20451.989} C_VEL
LIN {X 0,Y 232.318,Z 709.401,A -85,B 0,C 180,E1 -20453.866,E2 -20453.866} C_VEL
LIN {X 0,Y 234.171,Z 698.888,A -85,B 0,C 180,E1 -20455.311,E2 -20455.311} C_VEL
LIN {X 0,Y 236.001,Z 687.236,A -85,B 0,C 180,E1 -20456.531,E2 -20456.531} C_VEL
LIN {X 0,Y 237.297,Z 674.92,A -85,B 0,C 180,E1 -20457.493,E2 -20457.493} C_VEL
LIN {X 0,Y 238.268,Z 661.633,A -85,B 0,C 180,E1 -20458.16,E2 -20458.16} C_VEL
LIN {X 0,Y 241.082,Z 592.518,A -85,B 0,C 180,E1 -20460.156,E2 -20460.156} C_VEL
LIN {X 0,Y 238.606,Z 577.389,A -85,B 0,C 180,E1 -20461.044,E2 -20461.044} C_VEL
LIN {X 0,Y 233.161,Z 564.224,A -85,B 0,C 180,E1 -20462.365,E2 -20462.365} C_VEL
LIN {X 0,Y 227.081,Z 551.562,A -85,B 0,C 180,E1 -20463.925,E2 -20463.925} C_VEL
LIN {X 0,Y 223.812,Z 540.661,A -85,B 0,C 180,E1 -20467.66,E2 -20467.66} C_VEL
LIN {X 0,Y 220.839,Z 531.964,A -85,B 0,C 180,E1 -20470.987,E2 -20470.987} C_VEL
LIN {X 0,Y 220.855,Z 531.955,A -85,B 0,C 180,E1 -20474.748,E2 -20474.748} C_VEL
LIN {X 0,Y 231.562,Z 562.921,A -85,B 0,C 180,E1 -20477.054,E2 -20477.054} C_VEL
LIN {X 0,Y 228.441,Z 628.67,A -85,B 0,C 180,E1 -20479.971,E2 -20479.971} C_VEL
LIN {X 0,Y 227.593,Z 642.994,A -85,B 0,C 180,E1 -20480.981,E2 -20480.981} C_VEL
LIN {X 0,Y 226.427,Z 656.525,A -85,B 0,C 180,E1 -20482.332,E2 -20482.332} C_VEL
LIN {X 0,Y 225.212,Z 668.453,A -85,B 0,C 180,E1 -20483.882,E2 -20483.882} C_VEL
LIN {X 0,Y 223.836,Z 680.36,A -85,B 0,C 180,E1 -20485.858,E2 -20485.858} C_VEL
LIN {X 0,Y 222.639,Z 690.172,A -85,B 0,C 180,E1 -20487.876,E2 -20487.876} C_VEL
LIN {X 0,Y 221.577,Z 698.812,A -85,B 0,C 180,E1 -20490.028,E2 -20490.028} C_VEL
LIN {X 0,Y 220.6,Z 707.14,A -85,B 0,C 180,E1 -20492.556,E2 -20492.556} C_VEL
LIN {X 0,Y 219.811,Z 714.772,A -85,B 0,C 180,E1 -20495.439,E2 -20495.439} C_VEL
LIN {X 0,Y 219.228,Z 720.967,A -85,B 0,C 180,E1 -20498.381,E2 -20498.381} C_VEL
LIN {X 0,Y 218.938,Z 725.674,A -85,B 0,C 180,E1 -20501.276,E2 -20501.276} C_VEL
LIN {X 0,Y 218.987,Z 729.304,A -85,B 0,C 180,E1 -20504.317,E2 -20504.317} C_VEL
LIN {X 0,Y 219.34,Z 731.545,A -85,B 0,C 180,E1 -20507.038,E2 -20507.038} C_VEL
LIN {X 0,Y 219.803,Z 732.544,A -85,B 0,C 180,E1 -20508.939,E2 -20508.939} C_VEL
LIN {X 0,Y 220.536,Z 733.184,A -85,B 0,C 180,E1 -20511.07,E2 -20511.07} C_VEL
LIN {X 0,Y 221.244,Z 733.287,A -85,B 0,C 180,E1 -20512.7,E2 -20512.7} C_VEL
LIN {X 0,Y 222.391,Z 732.84,A -85,B 0,C 180,E1 -20514.905,E2 -20514.905} C_VEL
LIN {X 0,Y 222.682,Z 732.367,A -85,B 0,C 180,E1 -20516.419,E2 -20516.419} C_VEL
LIN {X 0,Y 221.701,Z 731.301,A -85,B 0,C 180,E1 -20518.952,E2 -20518.952} C_VEL
LIN {X 0,Y 221.093,Z 729.66,A -85,B 0,C 180,E1 -20521.474,E2 -20521.474} C_VEL
LIN {X 0,Y 221.942,Z 728.132,A -85,B 0,C 180,E1 -20522.931,E2 -20522.931} C_VEL
LIN {X 0,Y 224.871,Z 724.546,A -85,B 0,C 180,E1 -20525.38,E2 -20525.38} C_VEL
LIN {X 0,Y 228.443,Z 719.54,A -85,B 0,C 180,E1 -20527.957,E2 -20527.957} C_VEL
LIN {X 0,Y 233.268,Z 712.049,A -85,B 0,C 180,E1 -20530.853,E2 -20530.853} C_VEL
LIN {X 0,Y 237.768,Z 703.948,A -85,B 0,C 180,E1 -20533.242,E2 -20533.242} C_VEL
LIN {X 0,Y 241.849,Z 695.673,A -85,B 0,C 180,E1 -20535.161,E2 -20535.161} C_VEL
LIN {X 0,Y 246.213,Z 685.738,A -85,B 0,C 180,E1 -20537.012,E2 -20537.012} C_VEL
LIN {X 0,Y 250.324,Z 674.7,A -85,B 0,C 180,E1 -20538.624,E2 -20538.624} C_VEL
LIN {X 0,Y 254.139,Z 662.262,A -85,B 0,C 180,E1 -20540.039,E2 -20540.039} C_VEL
LIN {X 0,Y 257.229,Z 649.532,A -85,B 0,C 180,E1 -20541.144,E2 -20541.144} C_VEL
LIN {X 0,Y 259.61,Z 636.55,A -85,B 0,C 180,E1 -20541.981,E2 -20541.981} C_VEL
LIN {X 0,Y 263.719,Z 607.809,A -85,B 0,C 180,E1 -20543.231,E2 -20543.231} C_VEL
LIN {X 0,Y 265.034,Z 598.397,A -85,B 0,C 180,E1 -20543.653,E2 -20543.653} C_VEL
LIN {X 0,Y 262.207,Z 593.084,A -85,B 0,C 180,E1 -20545.844,E2 -20545.844} C_VEL
LIN {X 0,Y 259.864,Z 589.467,A -85,B 0,C 180,E1 -20548.02,E2 -20548.02} C_VEL
LIN {X 0,Y 258.026,Z 586.904,A -85,B 0,C 180,E1 -20550.25,E2 -20550.25} C_VEL
LIN {X 0,Y 256.089,Z 585.079,A -85,B 0,C 180,E1 -20553.961,E2 -20553.961} C_VEL
LIN {X 0,Y 255.625,Z 585.74,A -85,B 0,C 180,E1 -20556.877,E2 -20556.877} C_VEL
LIN {X 0,Y 256.078,Z 587.672,A -85,B 0,C 180,E1 -20559.69,E2 -20559.69} C_VEL
LIN {X 0,Y 258.003,Z 593.791,A -85,B 0,C 180,E1 -20563.704,E2 -20563.704} C_VEL
LIN {X 0,Y 260.212,Z 600.466,A -85,B 0,C 180,E1 -20566.431,E2 -20566.431} C_VEL
LIN {X 0,Y 262.306,Z 607.211,A -85,B 0,C 180,E1 -20568.456,E2 -20568.456} C_VEL
LIN {X 0,Y 262.807,Z 609.777,A -85,B 0,C 180,E1 -20569.011,E2 -20569.011} C_VEL
LIN {X 0,Y 262.494,Z 620.907,A -85,B 0,C 180,E1 -20570.049,E2 -20570.049} C_VEL
LIN {X 0,Y 261.803,Z 626.656,A -85,B 0,C 180,E1 -20570.342,E2 -20570.342} C_VEL
LIN {X 0,Y 257.297,Z 656.954,A -85,B 0,C 180,E1 -20571.644,E2 -20571.644} C_VEL
LIN {X 0,Y 254.271,Z 670.628,A -85,B 0,C 180,E1 -20572.426,E2 -20572.426} C_VEL
LIN {X 0,Y 250.583,Z 683.449,A -85,B 0,C 180,E1 -20573.418,E2 -20573.418} C_VEL
LIN {X 0,Y 246.301,Z 695.89,A -85,B 0,C 180,E1 -20574.704,E2 -20574.704} C_VEL
LIN {X 0,Y 241.228,Z 708.273,A -85,B 0,C 180,E1 -20576.39,E2 -20576.39} C_VEL
LIN {X 0,Y 236.554,Z 718.565,A -85,B 0,C 180,E1 -20578.174,E2 -20578.174} C_VEL
LIN {X 0,Y 231.529,Z 728.604,A -85,B 0,C 180,E1 -20580.445,E2 -20580.445} C_VEL
LIN {X 0,Y 226.999,Z 736.892,A -85,B 0,C 180,E1 -20582.828,E2 -20582.828} C_VEL
LIN {X 0,Y 223.077,Z 743.784,A -85,B 0,C 180,E1 -20585.328,E2 -20585.328} C_VEL
LIN {X 0,Y 219.294,Z 750.168,A -85,B 0,C 180,E1 -20588.341,E2 -20588.341} C_VEL
LIN {X 0,Y 215.739,Z 756.273,A -85,B 0,C 180,E1 -20592.218,E2 -20592.218} C_VEL
LIN {X 0,Y 214.118,Z 762.233,A -85,B 0,C 180,E1 -20594.777,E2 -20594.777} C_VEL
LIN {X 0,Y 212.815,Z 767.457,A -85,B 0,C 180,E1 -20597.605,E2 -20597.605} C_VEL
LIN {X 0,Y 212.043,Z 771.498,A -85,B 0,C 180,E1 -20600.461,E2 -20600.461} C_VEL
LIN {X 0,Y 211.722,Z 773.578,A -85,B 0,C 180,E1 -20602.37,E2 -20602.37} C_VEL
LIN {X 0,Y 211.485,Z 776.464,A -85,B 0,C 180,E1 -20606.189,E2 -20606.189} C_VEL
LIN {X 0,Y 211.488,Z 777.276,A -85,B 0,C 180,E1 -20608.096,E2 -20608.096} C_VEL
LIN {X 0,Y 211.555,Z 777.659,A -85,B 0,C 180,E1 -20610,E2 -20610} C_VEL
LIN {X 0,Y 211.485,Z 777.648,A -85,B 0,C 180,E1 -20611.904,E2 -20611.904} C_VEL
LIN {X 0,Y 211.473,Z 777.007,A -85,B 0,C 180,E1 -20614.434,E2 -20614.434} C_VEL
LIN {X 0,Y 211.719,Z 775.165,A -85,B 0,C 180,E1 -20617.63,E2 -20617.63} C_VEL
LIN {X 0,Y 212.339,Z 772.513,A -85,B 0,C 180,E1 -20620.488,E2 -20620.488} C_VEL
LIN {X 0,Y 213.266,Z 768.838,A -85,B 0,C 180,E1 -20623.337,E2 -20623.337} C_VEL
LIN {X 0,Y 214.824,Z 764.04,A -85,B 0,C 180,E1 -20626.145,E2 -20626.145} C_VEL
LIN {X 0,Y 216.789,Z 757.971,A -85,B 0,C 180,E1 -20628.916,E2 -20628.916} C_VEL
LIN {X 0,Y 219.169,Z 750.599,A -85,B 0,C 180,E1 -20631.576,E2 -20631.576} C_VEL
LIN {X 0,Y 221.558,Z 742.685,A -85,B 0,C 180,E1 -20633.855,E2 -20633.855} C_VEL
LIN {X 0,Y 224.36,Z 733.222,A -85,B 0,C 180,E1 -20636.01,E2 -20636.01} C_VEL
LIN {X 0,Y 227.192,Z 722.726,A -85,B 0,C 180,E1 -20637.896,E2 -20637.896} C_VEL
LIN {X 0,Y 229.509,Z 712.595,A -85,B 0,C 180,E1 -20639.337,E2 -20639.337} C_VEL
LIN {X 0,Y 231.82,Z 700.53,A -85,B 0,C 180,E1 -20640.643,E2 -20640.643} C_VEL
LIN {X 0,Y 233.828,Z 687.179,A -85,B 0,C 180,E1 -20641.67,E2 -20641.67} C_VEL
LIN {X 0,Y 235.105,Z 674.664,A -85,B 0,C 180,E1 -20642.298,E2 -20642.298} C_VEL
LIN {X 0,Y 237.623,Z 616.871,A -85,B 0,C 180,E1 -20644.006,E2 -20644.006} C_VEL
LIN {X 0,Y 234.729,Z 588.361,A -85,B 0,C 180,E1 -20645.552,E2 -20645.552} C_VEL
LIN {X 0,Y 233.25,Z 578.202,A -85,B 0,C 180,E1 -20646.202,E2 -20646.202} C_VEL
LIN {X 0,Y 226.985,Z 562.185,A -85,B 0,C 180,E1 -20648.039,E2 -20648.039} C_VEL
LIN {X 0,Y 225.274,Z 557.771,A -85,B 0,C 180,E1 -20648.604,E2 -20648.604} C_VEL
LIN {X 0,Y 223.644,Z 552.908,A -85,B 0,C 180,E1 -20649.778,E2 -20649.778} C_VEL
LIN {X 0,Y 218.178,Z 541.961,A -85,B 0,C 180,E1 -20652.978,E2 -20652.978} C_VEL
LIN {X 0,Y 213.947,Z 533.675,A -85,B 0,C 180,E1 -20655.731,E2 -20655.731} C_VEL
LIN {X 0,Y 213.777,Z 532.86,A -85,B 0,C 180,E1 -20656.047,E2 -20656.047} C_VEL
LIN {X 0,Y 213.749,Z 532.846,A -85,B 0,C 180,E1 -20659.132,E2 -20659.132} C_VEL
LIN {X 0,Y 213.751,Z 532.84,A -85,B 0,C 180,E1 -20663.713,E2 -20663.713} C_VEL
LIN {X 0,Y 213.776,Z 532.835,A -85,B 0,C 180,E1 -20668.264,E2 -20668.264} C_VEL
LIN {X 0,Y 213.822,Z 532.85,A -85,B 0,C 180,E1 -20672.603,E2 -20672.603} C_VEL
LIN {X 0,Y 213.815,Z 532.823,A -85,B 0,C 180,E1 -20676.974,E2 -20676.974} C_VEL
LIN {X 0,Y 213.938,Z 532.802,A -85,B 0,C 180,E1 -20682.803,E2 -20682.803} C_VEL
LIN {X 0,Y 213.973,Z 532.828,A -85,B 0,C 180,E1 -20686.708,E2 -20686.708} C_VEL
LIN {X 0,Y 214.162,Z 532.775,A -85,B 0,C 180,E1 -20690.557,E2 -20690.557} C_VEL
LIN {X 0,Y 214.222,Z 532.765,A -85,B 0,C 180,E1 -20692.46,E2 -20692.46} C_VEL
LIN {X 0,Y 214.442,Z 532.749,A -85,B 0,C 180,E1 -20698.122,E2 -20698.122} C_VEL
LIN {X 0,Y 214.545,Z 532.721,A -85,B 0,C 180,E1 -20700,E2 -20700} C_VEL
LIN {X 0,Y 214.442,Z 532.747,A -85,B 0,C 180,E1 -20701.879,E2 -20701.879} C_VEL
LIN {X 0,Y 214.194,Z 532.77,A -85,B 0,C 180,E1 -20707.542,E2 -20707.542} C_VEL
LIN {X 0,Y 213.994,Z 532.823,A -85,B 0,C 180,E1 -20711.365,E2 -20711.365} C_VEL
LIN {X 0,Y 213.925,Z 532.808,A -85,B 0,C 180,E1 -20715.238,E2 -20715.238} C_VEL
LIN {X 0,Y 213.864,Z 532.842,A -85,B 0,C 180,E1 -20719.186,E2 -20719.186} C_VEL
LIN {X 0,Y 213.844,Z 532.821,A -85,B 0,C 180,E1 -20723.228,E2 -20723.228} C_VEL
LIN {X 0,Y 213.827,Z 532.846,A -85,B 0,C 180,E1 -20727.451,E2 -20727.451} C_VEL
LIN {X 0,Y 213.775,Z 532.853,A -85,B 0,C 180,E1 -20731.737,E2 -20731.737} C_VEL
LIN {X 0,Y 213.742,Z 532.853,A -85,B 0,C 180,E1 -20736.289,E2 -20736.289} C_VEL
LIN {X 0,Y 213.759,Z 532.961,A -85,B 0,C 180,E1 -20740.425,E2 -20740.425} C_VEL
LIN {X 0,Y 217.894,Z 543.959,A -85,B 0,C 180,E1 -20745.203,E2 -20745.203} C_VEL
LIN {X 0,Y 220.629,Z 552.131,A -85,B 0,C 180,E1 -20748.373,E2 -20748.373} C_VEL
LIN {X 0,Y 227.65,Z 564.867,A -85,B 0,C 180,E1 -20750.38,E2 -20750.38} C_VEL
LIN {X 0,Y 234.3,Z 578.968,A -85,B 0,C 180,E1 -20752.201,E2 -20752.201} C_VEL
LIN {X 0,Y 237.588,Z 586.906,A -85,B 0,C 180,E1 -20753.084,E2 -20753.084} C_VEL
LIN {X 0,Y 239.014,Z 596.167,A -85,B 0,C 180,E1 -20753.667,E2 -20753.667} C_VEL
LIN {X 0,Y 235.841,Z 663.979,A -85,B 0,C 180,E1 -20755.645,E2 -20755.645} C_VEL
LIN {X 0,Y 234.594,Z 677.063,A -85,B 0,C 180,E1 -20756.344,E2 -20756.344} C_VEL
LIN {X 0,Y 232.891,Z 689.449,A -85,B 0,C 180,E1 -20757.345,E2 -20757.345} C_VEL
LIN {X 0,Y 230.718,Z 701.788,A -85,B 0,C 180,E1 -20758.715,E2 -20758.715} C_VEL
LIN {X 0,Y 228.09,Z 713.593,A -85,B 0,C 180,E1 -20760.463,E2 -20760.463} C_VEL
LIN {X 0,Y 225.363,Z 723.724,A -85,B 0,C 180,E1 -20762.363,E2 -20762.363} C_VEL
LIN {X 0,Y 222.859,Z 732.017,A -85,B 0,C 180,E1 -20764.304,E2 -20764.304} C_VEL
LIN {X 0,Y 219.932,Z 740.981,A -85,B 0,C 180,E1 -20766.956,E2 -20766.956} C_VEL
LIN {X 0,Y 217.55,Z 748.332,A -85,B 0,C 180,E1 -20769.747,E2 -20769.747} C_VEL
LIN {X 0,Y 215.397,Z 754.765,A -85,B 0,C 180,E1 -20772.924,E2 -20772.924} C_VEL
LIN {X 0,Y 213.769,Z 759.083,A -85,B 0,C 180,E1 -20775.725,E2 -20775.725} C_VEL
LIN {X 0,Y 212.733,Z 762.321,A -85,B 0,C 180,E1 -20778.567,E2 -20778.567} C_VEL
LIN {X 0,Y 212.233,Z 763.923,A -85,B 0,C 180,E1 -20780.47,E2 -20780.47} C_VEL
LIN {X 0,Y 211.852,Z 765.128,A -85,B 0,C 180,E1 -20782.375,E2 -20782.375} C_VEL
LIN {X 0,Y 211.484,Z 766.219,A -85,B 0,C 180,E1 -20785.536,E2 -20785.536} C_VEL
LIN {X 0,Y 211.489,Z 766.271,A -85,B 0,C 180,E1 -20788.096,E2 -20788.096} C_VEL
LIN {X 0,Y 211.555,Z 765.883,A -85,B 0,C 180,E1 -20790,E2 -20790} C_VEL
LIN {X 0,Y 211.66,Z 765.07,A -85,B 0,C 180,E1 -20791.903,E2 -20791.903} C_VEL
LIN {X 0,Y 211.94,Z 763.85,A -85,B 0,C 180,E1 -20793.803,E2 -20793.803} C_VEL
LIN {X 0,Y 212.383,Z 761.58,A -85,B 0,C 180,E1 -20796.355,E2 -20796.355} C_VEL
LIN {X 0,Y 213.315,Z 757.659,A -85,B 0,C 180,E1 -20799.481,E2 -20799.481} C_VEL
LIN {X 0,Y 214.599,Z 752.95,A -85,B 0,C 180,E1 -20802.29,E2 -20802.29} C_VEL
LIN {X 0,Y 216.281,Z 746.993,A -85,B 0,C 180,E1 -20805.067,E2 -20805.067} C_VEL
LIN {X 0,Y 218.45,Z 739.571,A -85,B 0,C 180,E1 -20807.796,E2 -20807.796} C_VEL
LIN {X 0,Y 220.906,Z 730.226,A -85,B 0,C 180,E1 -20810.484,E2 -20810.484} C_VEL
LIN {X 0,Y 223.381,Z 720.594,A -85,B 0,C 180,E1 -20812.669,E2 -20812.669} C_VEL
LIN {X 0,Y 225.867,Z 709.781,A -85,B 0,C 180,E1 -20814.592,E2 -20814.592} C_VEL
LIN {X 0,Y 228.048,Z 697.844,A -85,B 0,C 180,E1 -20816.253,E2 -20816.253} C_VEL
LIN {X 0,Y 229.823,Z 686.729,A -85,B 0,C 180,E1 -20817.416,E2 -20817.416} C_VEL
LIN {X 0,Y 231.145,Z 674.632,A -85,B 0,C 180,E1 -20818.358,E2 -20818.358} C_VEL
LIN {X 0,Y 232.19,Z 660.627,A -85,B 0,C 180,E1 -20819.054,E2 -20819.054} C_VEL
LIN {X 0,Y 234.985,Z 593.285,A -85,B 0,C 180,E1 -20821.036,E2 -20821.036} C_VEL
LIN {X 0,Y 232.751,Z 579.78,A -85,B 0,C 180,E1 -20821.869,E2 -20821.869} C_VEL
LIN {X 0,Y 227.197,Z 566.258,A -85,B 0,C 180,E1 -20823.29,E2 -20823.29} C_VEL
LIN {X 0,Y 220.011,Z 551.806,A -85,B 0,C 180,E1 -20825.189,E2 -20825.189} C_VEL
LIN {X 0,Y 216.842,Z 541.409,A -85,B 0,C 180,E1 -20828.934,E2 -20828.934} C_VEL
LIN {X 0,Y 213.82,Z 532.852,A -85,B 0,C 180,E1 -20832.416,E2 -20832.416} C_VEL
LIN {X 0,Y 213.819,Z 532.834,A -85,B 0,C 180,E1 -20834.256,E2 -20834.256} C_VEL
LIN {X 0,Y 224.525,Z 563.786,A -85,B 0,C 180,E1 -20836.615,E2 -20836.615} C_VEL
LIN {X 0,Y 221.447,Z 629.256,A -85,B 0,C 180,E1 -20839.646,E2 -20839.646} C_VEL
LIN {X 0,Y 220.594,Z 643.727,A -85,B 0,C 180,E1 -20840.712,E2 -20840.712} C_VEL
LIN {X 0,Y 219.383,Z 656.847,A -85,B 0,C 180,E1 -20842.071,E2 -20842.071} C_VEL
LIN {X 0,Y 218.181,Z 668.529,A -85,B 0,C 180,E1 -20843.637,E2 -20843.637} C_VEL
LIN {X 0,Y 216.757,Z 680.7,A -85,B 0,C 180,E1 -20845.711,E2 -20845.711} C_VEL
LIN {X 0,Y 215.362,Z 691.645,A -85,B 0,C 180,E1 -20848.043,E2 -20848.043} C_VEL
LIN {X 0,Y 214.233,Z 700.984,A -85,B 0,C 180,E1 -20850.522,E2 -20850.522} C_VEL
LIN {X 0,Y 213.174,Z 710.249,A -85,B 0,C 180,E1 -20853.571,E2 -20853.571} C_VEL
LIN {X 0,Y 212.457,Z 717.506,A -85,B 0,C 180,E1 -20856.611,E2 -20856.611} C_VEL
LIN {X 0,Y 212,Z 723.159,A -85,B 0,C 180,E1 -20859.629,E2 -20859.629} C_VEL
LIN {X 0,Y 211.801,Z 727.464,A -85,B 0,C 180,E1 -20862.624,E2 -20862.624} C_VEL
LIN {X 0,Y 211.928,Z 729.708,A -85,B 0,C 180,E1 -20864.615,E2 -20864.615} C_VEL
LIN {X 0,Y 212.179,Z 731.415,A -85,B 0,C 180,E1 -20866.593,E2 -20866.593} C_VEL
LIN {X 0,Y 212.6,Z 732.694,A -85,B 0,C 180,E1 -20868.559,E2 -20868.559} C_VEL
LIN {X 0,Y 213.427,Z 733.67,A -85,B 0,C 180,E1 -20871.061,E2 -20871.061} C_VEL
LIN {X 0,Y 214.96,Z 733.865,A -85,B 0,C 180,E1 -20874.371,E2 -20874.371} C_VEL
LIN {X 0,Y 216.128,Z 733.417,A -85,B 0,C 180,E1 -20876.271,E2 -20876.271} C_VEL
LIN {X 0,Y 217.919,Z 732.167,A -85,B 0,C 180,E1 -20878.697,E2 -20878.697} C_VEL
LIN {X 0,Y 220.753,Z 729.443,A -85,B 0,C 180,E1 -20881.824,E2 -20881.824} C_VEL
LIN {X 0,Y 221.942,Z 728.132,A -85,B 0,C 180,E1 -20882.931,E2 -20882.931} C_VEL
LIN {X 0,Y 222.927,Z 726.415,A -85,B 0,C 180,E1 -20884.367,E2 -20884.367} C_VEL
LIN {X 0,Y 223.153,Z 723.575,A -85,B 0,C 180,E1 -20886.812,E2 -20886.812} C_VEL
LIN {X 0,Y 223.723,Z 720.125,A -85,B 0,C 180,E1 -20889.181,E2 -20889.181} C_VEL
LIN {X 0,Y 225.19,Z 717.45,A -85,B 0,C 180,E1 -20890.463,E2 -20890.463} C_VEL
LIN {X 0,Y 229.55,Z 710.807,A -85,B 0,C 180,E1 -20892.825,E2 -20892.825} C_VEL
LIN {X 0,Y 234.445,Z 702.339,A -85,B 0,C 180,E1 -20895.206,E2 -20895.206} C_VEL
LIN {X 0,Y 238.906,Z 693.624,A -85,B 0,C 180,E1 -20897.108,E2 -20897.108} C_VEL
LIN {X 0,Y 243.605,Z 682.994,A -85,B 0,C 180,E1 -20898.939,E2 -20898.939} C_VEL
LIN {X 0,Y 247.71,Z 672.096,A -85,B 0,C 180,E1 -20900.426,E2 -20900.426} C_VEL
LIN {X 0,Y 251.62,Z 659.423,A -85,B 0,C 180,E1 -20901.774,E2 -20901.774} C_VEL
LIN {X 0,Y 254.61,Z 646.797,A -85,B 0,C 180,E1 -20902.79,E2 -20902.79} C_VEL
LIN {X 0,Y 256.655,Z 635.469,A -85,B 0,C 180,E1 -20903.45,E2 -20903.45} C_VEL
LIN {X 0,Y 260.505,Z 610.126,A -85,B 0,C 180,E1 -20904.567,E2 -20904.567} C_VEL
LIN {X 0,Y 261.665,Z 602.845,A -85,B 0,C 180,E1 -20904.866,E2 -20904.866} C_VEL
LIN {X 0,Y 259.644,Z 598.938,A -85,B 0,C 180,E1 -20906.611,E2 -20906.611} C_VEL
LIN {X 0,Y 257.867,Z 596.083,A -85,B 0,C 180,E1 -20908.41,E2 -20908.41} C_VEL
LIN {X 0,Y 256.484,Z 593.871,A -85,B 0,C 180,E1 -20910.231,E2 -20910.231} C_VEL
LIN {X 0,Y 254.53,Z 592.003,A -85,B 0,C 180,E1 -20914.072,E2 -20914.072} C_VEL
LIN {X 0,Y 254.078,Z 592.606,A -85,B 0,C 180,E1 -20916.665,E2 -20916.665} C_VEL
LIN {X 0,Y 254.398,Z 594.377,A -85,B 0,C 180,E1 -20919.33,E2 -20919.33} C_VEL
LIN {X 0,Y 255.931,Z 599.965,A -85,B 0,C 180,E1 -20923.037,E2 -20923.037} C_VEL
LIN {X 0,Y 257.868,Z 606.501,A -85,B 0,C 180,E1 -20925.773,E2 -20925.773} C_VEL
LIN {X 0,Y 259.163,Z 611.268,A -85,B 0,C 180,E1 -20927.258,E2 -20927.258} C_VEL
LIN {X 0,Y 259.687,Z 613.689,A -85,B 0,C 180,E1 -20927.86,E2 -20927.86} C_VEL
LIN {X 0,Y 259.145,Z 623.507,A -85,B 0,C 180,E1 -20928.791,E2 -20928.791} C_VEL
LIN {X 0,Y 254.09,Z 656.248,A -85,B 0,C 180,E1 -20930.198,E2 -20930.198} C_VEL
LIN {X 0,Y 250.706,Z 670.58,A -85,B 0,C 180,E1 -20931.026,E2 -20931.026} C_VEL
LIN {X 0,Y 246.28,Z 684.818,A -85,B 0,C 180,E1 -20932.155,E2 -20932.155} C_VEL
LIN {X 0,Y 240.717,Z 699.395,A -85,B 0,C 180,E1 -20933.757,E2 -20933.757} C_VEL
LIN {X 0,Y 235.525,Z 710.975,A -85,B 0,C 180,E1 -20935.463,E2 -20935.463} C_VEL
LIN {X 0,Y 230.706,Z 720.538,A -85,B 0,C 180,E1 -20937.268,E2 -20937.268} C_VEL
LIN {X 0,Y 225.506,Z 730.104,A -85,B 0,C 180,E1 -20939.574,E2 -20939.574} C_VEL
LIN {X 0,Y 220.786,Z 737.979,A -85,B 0,C 180,E1 -20941.998,E2 -20941.998} C_VEL
LIN {X 0,Y 217.347,Z 743.487,A -85,B 0,C 180,E1 -20944.118,E2 -20944.118} C_VEL
LIN {X 0,Y 213.743,Z 749.019,A -85,B 0,C 180,E1 -20946.762,E2 -20946.762} C_VEL
LIN {X 0,Y 210.821,Z 753.473,A -85,B 0,C 180,E1 -20949.511,E2 -20949.511} C_VEL
LIN {X 0,Y 208.777,Z 756.619,A -85,B 0,C 180,E1 -20951.858,E2 -20951.858} C_VEL
LIN {X 0,Y 207.266,Z 761.98,A -85,B 0,C 180,E1 -20954.261,E2 -20954.261} C_VEL
LIN {X 0,Y 205.857,Z 767.215,A -85,B 0,C 180,E1 -20957.179,E2 -20957.179} C_VEL
LIN {X 0,Y 204.997,Z 771.268,A -85,B 0,C 180,E1 -20960.13,E2 -20960.13} C_VEL
LIN {X 0,Y 204.665,Z 773.359,A -85,B 0,C 180,E1 -20962.105,E2 -20962.105} C_VEL
LIN {X 0,Y 204.378,Z 776.07,A -85,B 0,C 180,E1 -20965.734,E2 -20965.734} C_VEL
LIN {X 0,Y 204.392,Z 777.077,A -85,B 0,C 180,E1 -20968.03,E2 -20968.03} C_VEL
LIN {X 0,Y 204.474,Z 777.466,A -85,B 0,C 180,E1 -20970,E2 -20970} C_VEL
LIN {X 0,Y 204.388,Z 777.46,A -85,B 0,C 180,E1 -20971.97,E2 -20971.97} C_VEL
LIN {X 0,Y 204.384,Z 776.952,A -85,B 0,C 180,E1 -20974.287,E2 -20974.287} C_VEL
LIN {X 0,Y 204.663,Z 774.997,A -85,B 0,C 180,E1 -20977.895,E2 -20977.895} C_VEL
LIN {X 0,Y 205.317,Z 772.355,A -85,B 0,C 180,E1 -20980.851,E2 -20980.851} C_VEL
LIN {X 0,Y 206.32,Z 768.692,A -85,B 0,C 180,E1 -20983.794,E2 -20983.794} C_VEL
LIN {X 0,Y 207.979,Z 763.907,A -85,B 0,C 180,E1 -20986.692,E2 -20986.692} C_VEL
LIN {X 0,Y 210.066,Z 757.853,A -85,B 0,C 180,E1 -20989.545,E2 -20989.545} C_VEL
LIN {X 0,Y 212.716,Z 750.038,A -85,B 0,C 180,E1 -20992.434,E2 -20992.434} C_VEL
LIN {X 0,Y 215.618,Z 740.848,A -85,B 0,C 180,E1 -20995.07,E2 -20995.07} C_VEL
LIN {X 0,Y 218.63,Z 731.061,A -85,B 0,C 180,E1 -20997.262,E2 -20997.262} C_VEL
LIN {X 0,Y 221.573,Z 720.037,A -85,B 0,C 180,E1 -20999.187,E2 -20999.187} C_VEL
LIN {X 0,Y 224.039,Z 709.244,A -85,B 0,C 180,E1 -21000.647,E2 -21000.647} C_VEL
LIN {X 0,Y 226.3,Z 697.34,A -85,B 0,C 180,E1 -21001.866,E2 -21001.866} C_VEL
LIN {X 0,Y 228.098,Z 685.048,A -85,B 0,C 180,E1 -21002.759,E2 -21002.759} C_VEL
LIN {X 0,Y 229.31,Z 672.464,A -85,B 0,C 180,E1 -21003.349,E2 -21003.349} C_VEL
LIN {X 0,Y 231.801,Z 618.091,A -85,B 0,C 180,E1 -21004.969,E2 -21004.969} C_VEL
LIN {X 0,Y 229.286,Z 591.516,A -85,B 0,C 180,E1 -21006.439,E2 -21006.439} C_VEL
LIN {X 0,Y 227.695,Z 580.489,A -85,B 0,C 180,E1 -21007.175,E2 -21007.175} C_VEL
LIN {X 0,Y 220.044,Z 560.874,A -85,B 0,C 180,E1 -21009.568,E2 -21009.568} C_VEL
LIN {X 0,Y 218.591,Z 557.992,A -85,B 0,C 180,E1 -21010.017,E2 -21010.017} C_VEL
LIN {X 0,Y 213.06,Z 546.51,A -85,B 0,C 180,E1 -21013.474,E2 -21013.474} C_VEL
LIN {X 0,Y 209.003,Z 538.376,A -85,B 0,C 180,E1 -21016.261,E2 -21016.261} C_VEL
LIN {X 0,Y 207.313,Z 535.878,A -85,B 0,C 180,E1 -21017.312,E2 -21017.312} C_VEL
LIN {X 0,Y 206.681,Z 533.724,A -85,B 0,C 180,E1 -21018.048,E2 -21018.048} C_VEL
LIN {X 0,Y 206.718,Z 533.72,A -85,B 0,C 180,E1 -21022.269,E2 -21022.269} C_VEL
LIN {X 0,Y 206.706,Z 533.731,A -85,B 0,C 180,E1 -21027.044,E2 -21027.044} C_VEL
LIN {X 0,Y 206.763,Z 533.729,A -85,B 0,C 180,E1 -21032.096,E2 -21032.096} C_VEL
LIN {X 0,Y 206.749,Z 533.7,A -85,B 0,C 180,E1 -21036.604,E2 -21036.604} C_VEL
LIN {X 0,Y 206.868,Z 533.687,A -85,B 0,C 180,E1 -21042.196,E2 -21042.196} C_VEL
LIN {X 0,Y 206.906,Z 533.703,A -85,B 0,C 180,E1 -21046.245,E2 -21046.245} C_VEL
LIN {X 0,Y 207.101,Z 533.657,A -85,B 0,C 180,E1 -21050.231,E2 -21050.231} C_VEL
LIN {X 0,Y 207.163,Z 533.642,A -85,B 0,C 180,E1 -21052.201,E2 -21052.201} C_VEL
LIN {X 0,Y 207.378,Z 533.629,A -85,B 0,C 180,E1 -21058.058,E2 -21058.058} C_VEL
LIN {X 0,Y 207.51,Z 533.596,A -85,B 0,C 180,E1 -21060,E2 -21060} C_VEL
LIN {X 0,Y 207.379,Z 533.626,A -85,B 0,C 180,E1 -21061.943,E2 -21061.943} C_VEL
LIN {X 0,Y 207.137,Z 533.647,A -85,B 0,C 180,E1 -21067.801,E2 -21067.801} C_VEL
LIN {X 0,Y 206.92,Z 533.709,A -85,B 0,C 180,E1 -21071.759,E2 -21071.759} C_VEL
LIN {X 0,Y 206.859,Z 533.685,A -85,B 0,C 180,E1 -21075.772,E2 -21075.772} C_VEL
LIN {X 0,Y 206.796,Z 533.726,A -85,B 0,C 180,E1 -21079.868,E2 -21079.868} C_VEL
LIN {X 0,Y 206.761,Z 533.705,A -85,B 0,C 180,E1 -21084.073,E2 -21084.073} C_VEL
LIN {X 0,Y 206.742,Z 533.715,A -85,B 0,C 180,E1 -21088.42,E2 -21088.42} C_VEL
LIN {X 0,Y 206.7,Z 533.736,A -85,B 0,C 180,E1 -21092.958,E2 -21092.958} C_VEL
LIN {X 0,Y 206.679,Z 533.743,A -85,B 0,C 180,E1 -21097.741,E2 -21097.741} C_VEL
LIN {X 0,Y 206.694,Z 533.875,A -85,B 0,C 180,E1 -21098.51,E2 -21098.51} C_VEL
LIN {X 0,Y 210.546,Z 543.759,A -85,B 0,C 180,E1 -21103.179,E2 -21103.179} C_VEL
LIN {X 0,Y 213.701,Z 552.527,A -85,B 0,C 180,E1 -21106.775,E2 -21106.775} C_VEL
LIN {X 0,Y 221.94,Z 567.249,A -85,B 0,C 180,E1 -21109.29,E2 -21109.29} C_VEL
LIN {X 0,Y 227.253,Z 578.224,A -85,B 0,C 180,E1 -21110.829,E2 -21110.829} C_VEL
LIN {X 0,Y 232.06,Z 589.535,A -85,B 0,C 180,E1 -21112.188,E2 -21112.188} C_VEL
LIN {X 0,Y 233.196,Z 597.056,A -85,B 0,C 180,E1 -21112.68,E2 -21112.68} C_VEL
LIN {X 0,Y 229.926,Z 664.64,A -85,B 0,C 180,E1 -21114.698,E2 -21114.698} C_VEL
LIN {X 0,Y 228.622,Z 677.509,A -85,B 0,C 180,E1 -21115.408,E2 -21115.408} C_VEL
LIN {X 0,Y 226.881,Z 689.614,A -85,B 0,C 180,E1 -21116.406,E2 -21116.406} C_VEL
LIN {X 0,Y 224.806,Z 700.858,A -85,B 0,C 180,E1 -21117.659,E2 -21117.659} C_VEL
LIN {X 0,Y 222.267,Z 712.331,A -85,B 0,C 180,E1 -21119.346,E2 -21119.346} C_VEL
LIN {X 0,Y 219.349,Z 722.709,A -85,B 0,C 180,E1 -21121.276,E2 -21121.276} C_VEL
LIN {X 0,Y 216.461,Z 732.074,A -85,B 0,C 180,E1 -21123.486,E2 -21123.486} C_VEL
LIN {X 0,Y 213.395,Z 741.071,A -85,B 0,C 180,E1 -21126.207,E2 -21126.207} C_VEL
LIN {X 0,Y 210.722,Z 748.875,A -85,B 0,C 180,E1 -21129.264,E2 -21129.264} C_VEL
LIN {X 0,Y 208.597,Z 754.897,A -85,B 0,C 180,E1 -21132.349,E2 -21132.349} C_VEL
LIN {X 0,Y 206.862,Z 759.229,A -85,B 0,C 180,E1 -21135.238,E2 -21135.238} C_VEL
LIN {X 0,Y 205.761,Z 762.48,A -85,B 0,C 180,E1 -21138.174,E2 -21138.174} C_VEL
LIN {X 0,Y 204.805,Z 765.299,A -85,B 0,C 180,E1 -21142.111,E2 -21142.111} C_VEL
LIN {X 0,Y 204.414,Z 766.436,A -85,B 0,C 180,E1 -21145.613,E2 -21145.613} C_VEL
LIN {X 0,Y 204.393,Z 766.465,A -85,B 0,C 180,E1 -21148.03,E2 -21148.03} C_VEL
LIN {X 0,Y 204.474,Z 766.082,A -85,B 0,C 180,E1 -21150,E2 -21150} C_VEL
LIN {X 0,Y 204.585,Z 765.281,A -85,B 0,C 180,E1 -21151.969,E2 -21151.969} C_VEL
LIN {X 0,Y 204.876,Z 764.067,A -85,B 0,C 180,E1 -21153.934,E2 -21153.934} C_VEL
LIN {X 0,Y 205.568,Z 760.837,A -85,B 0,C 180,E1 -21157.489,E2 -21157.489} C_VEL
LIN {X 0,Y 206.718,Z 756.487,A -85,B 0,C 180,E1 -21160.777,E2 -21160.777} C_VEL
LIN {X 0,Y 208.226,Z 751.385,A -85,B 0,C 180,E1 -21163.666,E2 -21163.666} C_VEL
LIN {X 0,Y 210.498,Z 743.761,A -85,B 0,C 180,E1 -21166.986,E2 -21166.986} C_VEL
LIN {X 0,Y 212.991,Z 735.462,A -85,B 0,C 180,E1 -21169.768,E2 -21169.768} C_VEL
LIN {X 0,Y 215.281,Z 726.928,A -85,B 0,C 180,E1 -21172.05,E2 -21172.05} C_VEL
LIN {X 0,Y 217.972,Z 716.447,A -85,B 0,C 180,E1 -21174.273,E2 -21174.273} C_VEL
LIN {X 0,Y 220.379,Z 705.973,A -85,B 0,C 180,E1 -21176.007,E2 -21176.007} C_VEL
LIN {X 0,Y 222.34,Z 695.177,A -85,B 0,C 180,E1 -21177.418,E2 -21177.418} C_VEL
LIN {X 0,Y 224.103,Z 682.94,A -85,B 0,C 180,E1 -21178.631,E2 -21178.631} C_VEL
LIN {X 0,Y 225.43,Z 670.008,A -85,B 0,C 180,E1 -21179.535,E2 -21179.535} C_VEL
LIN {X 0,Y 226.321,Z 656.177,A -85,B 0,C 180,E1 -21180.105,E2 -21180.105} C_VEL
LIN {X 0,Y 228.927,Z 594.244,A -85,B 0,C 180,E1 -21181.959,E2 -21181.959} C_VEL
LIN {X 0,Y 227.079,Z 582.419,A -85,B 0,C 180,E1 -21182.704,E2 -21182.704} C_VEL
LIN {X 0,Y 221.337,Z 568.652,A -85,B 0,C 180,E1 -21184.241,E2 -21184.241} C_VEL
LIN {X 0,Y 214.701,Z 555.439,A -85,B 0,C 180,E1 -21186.05,E2 -21186.05} C_VEL
LIN {X 0,Y 212.969,Z 552.04,A -85,B 0,C 180,E1 -21186.571,E2 -21186.571} C_VEL
LIN {X 0,Y 209.799,Z 542.242,A -85,B 0,C 180,E1 -21190.293,E2 -21190.293} C_VEL
LIN {X 0,Y 206.821,Z 533.986,A -85,B 0,C 180,E1 -21193.769,E2 -21193.769} C_VEL
LIN {X 0,Y 217.671,Z 565.384,A -85,B 0,C 180,E1 -21196.227,E2 -21196.227} C_VEL
LIN {X 0,Y 214.418,Z 630.049,A -85,B 0,C 180,E1 -21199.349,E2 -21199.349} C_VEL
LIN {X 0,Y 213.613,Z 643.824,A -85,B 0,C 180,E1 -21200.397,E2 -21200.397} C_VEL
LIN {X 0,Y 212.365,Z 657.069,A -85,B 0,C 180,E1 -21201.798,E2 -21201.798} C_VEL
LIN {X 0,Y 211.072,Z 669.206,A -85,B 0,C 180,E1 -21203.474,E2 -21203.474} C_VEL
LIN {X 0,Y 209.686,Z 681.045,A -85,B 0,C 180,E1 -21205.555,E2 -21205.555} C_VEL
LIN {X 0,Y 208.291,Z 691.752,A -85,B 0,C 180,E1 -21207.898,E2 -21207.898} C_VEL
LIN {X 0,Y 207.089,Z 701.41,A -85,B 0,C 180,E1 -21210.521,E2 -21210.521} C_VEL
LIN {X 0,Y 206.255,Z 708.724,A -85,B 0,C 180,E1 -21212.956,E2 -21212.956} C_VEL
LIN {X 0,Y 205.521,Z 715.681,A -85,B 0,C 180,E1 -21215.772,E2 -21215.772} C_VEL
LIN {X 0,Y 204.976,Z 721.879,A -85,B 0,C 180,E1 -21218.898,E2 -21218.898} C_VEL
LIN {X 0,Y 204.728,Z 726.674,A -85,B 0,C 180,E1 -21222.003,E2 -21222.003} C_VEL
LIN {X 0,Y 204.875,Z 730.245,A -85,B 0,C 180,E1 -21225.091,E2 -21225.091} C_VEL
LIN {X 0,Y 205.388,Z 732.709,A -85,B 0,C 180,E1 -21228.152,E2 -21228.152} C_VEL
LIN {X 0,Y 206.318,Z 734.106,A -85,B 0,C 180,E1 -21231.052,E2 -21231.052} C_VEL
LIN {X 0,Y 207.719,Z 734.632,A -85,B 0,C 180,E1 -21234.174,E2 -21234.174} C_VEL
LIN {X 0,Y 208.892,Z 734.423,A -85,B 0,C 180,E1 -21236.141,E2 -21236.141} C_VEL
LIN {X 0,Y 211.849,Z 732.722,A -85,B 0,C 180,E1 -21240,E2 -21240} C_VEL
LIN {X 0,Y 213.622,Z 731.27,A -85,B 0,C 180,E1 -21241.885,E2 -21241.885} C_VEL
LIN {X 0,Y 216.717,Z 728.195,A -85,B 0,C 180,E1 -21244.65,E2 -21244.65} C_VEL
LIN {X 0,Y 220.225,Z 724.072,A -85,B 0,C 180,E1 -21247.334,E2 -21247.334} C_VEL
LIN {X 0,Y 224.985,Z 717.74,A -85,B 0,C 180,E1 -21250.347,E2 -21250.347} C_VEL
LIN {X 0,Y 225.19,Z 717.45,A -85,B 0,C 180,E1 -21250.463,E2 -21250.463} C_VEL
LIN {X 0,Y 226.763,Z 714.601,A -85,B 0,C 180,E1 -21251.716,E2 -21251.716} C_VEL
LIN {X 0,Y 227.985,Z 710.069,A -85,B 0,C 180,E1 -21253.921,E2 -21253.921} C_VEL
LIN {X 0,Y 229.377,Z 705.016,A -85,B 0,C 180,E1 -21256.014,E2 -21256.014} C_VEL
LIN {X 0,Y 231.134,Z 701.33,A -85,B 0,C 180,E1 -21257.065,E2 -21257.065} C_VEL
LIN {X 0,Y 236.303,Z 691.574,A -85,B 0,C 180,E1 -21259.096,E2 -21259.096} C_VEL
LIN {X 0,Y 241.031,Z 681.096,A -85,B 0,C 180,E1 -21260.796,E2 -21260.796} C_VEL
LIN {X 0,Y 245.472,Z 669.329,A -85,B 0,C 180,E1 -21262.294,E2 -21262.294} C_VEL
LIN {X 0,Y 249.144,Z 657.357,A -85,B 0,C 180,E1 -21263.481,E2 -21263.481} C_VEL
LIN {X 0,Y 252.362,Z 644.023,A -85,B 0,C 180,E1 -21264.472,E2 -21264.472} C_VEL
LIN {X 0,Y 255.159,Z 627.262,A -85,B 0,C 180,E1 -21265.333,E2 -21265.333} C_VEL
LIN {X 0,Y 258.409,Z 607.152,A -85,B 0,C 180,E1 -21266.17,E2 -21266.17} C_VEL
LIN {X 0,Y 256.098,Z 602.922,A -85,B 0,C 180,E1 -21268.581,E2 -21268.581} C_VEL
LIN {X 0,Y 254.751,Z 600.676,A -85,B 0,C 180,E1 -21270.458,E2 -21270.458} C_VEL
LIN {X 0,Y 253.076,Z 598.999,A -85,B 0,C 180,E1 -21273.738,E2 -21273.738} C_VEL
LIN {X 0,Y 252.535,Z 599.497,A -85,B 0,C 180,E1 -21276.501,E2 -21276.501} C_VEL
LIN {X 0,Y 252.738,Z 601.195,A -85,B 0,C 180,E1 -21279.039,E2 -21279.039} C_VEL
LIN {X 0,Y 254.085,Z 606.683,A -85,B 0,C 180,E1 -21282.696,E2 -21282.696} C_VEL
LIN {X 0,Y 255.584,Z 612.609,A -85,B 0,C 180,E1 -21285.138,E2 -21285.138} C_VEL
LIN {X 0,Y 256.692,Z 617.622,A -85,B 0,C 180,E1 -21286.685,E2 -21286.685} C_VEL
LIN {X 0,Y 256.209,Z 625.156,A -85,B 0,C 180,E1 -21287.406,E2 -21287.406} C_VEL
LIN {X 0,Y 251.201,Z 655.324,A -85,B 0,C 180,E1 -21288.694,E2 -21288.694} C_VEL
LIN {X 0,Y 247.614,Z 669.677,A -85,B 0,C 180,E1 -21289.515,E2 -21289.515} C_VEL
LIN {X 0,Y 243.302,Z 683.109,A -85,B 0,C 180,E1 -21290.545,E2 -21290.545} C_VEL
LIN {X 0,Y 238.628,Z 695.152,A -85,B 0,C 180,E1 -21291.795,E2 -21291.795} C_VEL
LIN {X 0,Y 233.585,Z 706.197,A -85,B 0,C 180,E1 -21293.275,E2 -21293.275} C_VEL
LIN {X 0,Y 227.851,Z 717.342,A -85,B 0,C 180,E1 -21295.207,E2 -21295.207} C_VEL
LIN {X 0,Y 222.182,Z 727.258,A -85,B 0,C 180,E1 -21297.471,E2 -21297.471} C_VEL
LIN {X 0,Y 217.008,Z 735.441,A -85,B 0,C 180,E1 -21299.87,E2 -21299.87} C_VEL
LIN {X 0,Y 212.402,Z 742.268,A -85,B 0,C 180,E1 -21302.405,E2 -21302.405} C_VEL
LIN {X 0,Y 208.434,Z 747.848,A -85,B 0,C 180,E1 -21305.073,E2 -21305.073} C_VEL
LIN {X 0,Y 205.155,Z 752.346,A -85,B 0,C 180,E1 -21307.863,E2 -21307.863} C_VEL
LIN {X 0,Y 201.86,Z 756.649,A -85,B 0,C 180,E1 -21311.345,E2 -21311.345} C_VEL
LIN {X 0,Y 200.393,Z 761.725,A -85,B 0,C 180,E1 -21313.706,E2 -21313.706} C_VEL
LIN {X 0,Y 198.889,Z 766.972,A -85,B 0,C 180,E1 -21316.722,E2 -21316.722} C_VEL
LIN {X 0,Y 197.971,Z 771.037,A -85,B 0,C 180,E1 -21319.776,E2 -21319.776} C_VEL
LIN {X 0,Y 197.606,Z 773.139,A -85,B 0,C 180,E1 -21321.821,E2 -21321.821} C_VEL
LIN {X 0,Y 197.366,Z 774.794,A -85,B 0,C 180,E1 -21323.868,E2 -21323.868} C_VEL
LIN {X 0,Y 197.285,Z 776.045,A -85,B 0,C 180,E1 -21325.914,E2 -21325.914} C_VEL
LIN {X 0,Y 197.297,Z 776.878,A -85,B 0,C 180,E1 -21327.959,E2 -21327.959} C_VEL
LIN {X 0,Y 197.375,Z 777.272,A -85,B 0,C 180,E1 -21330,E2 -21330} C_VEL
LIN {X 0,Y 197.294,Z 777.271,A -85,B 0,C 180,E1 -21332.041,E2 -21332.041} C_VEL
LIN {X 0,Y 197.285,Z 776.881,A -85,B 0,C 180,E1 -21334.086,E2 -21334.086} C_VEL
LIN {X 0,Y 197.365,Z 776.068,A -85,B 0,C 180,E1 -21336.132,E2 -21336.132} C_VEL
LIN {X 0,Y 198.04,Z 773.188,A -85,B 0,C 180,E1 -21340.22,E2 -21340.22} C_VEL
LIN {X 0,Y 199.003,Z 769.885,A -85,B 0,C 180,E1 -21343.27,E2 -21343.27} C_VEL
LIN {X 0,Y 200.521,Z 765.505,A -85,B 0,C 180,E1 -21346.283,E2 -21346.283} C_VEL
LIN {X 0,Y 202.601,Z 759.921,A -85,B 0,C 180,E1 -21349.241,E2 -21349.241} C_VEL
LIN {X 0,Y 205.141,Z 752.915,A -85,B 0,C 180,E1 -21352.138,E2 -21352.138} C_VEL
LIN {X 0,Y 208.06,Z 744.161,A -85,B 0,C 180,E1 -21354.975,E2 -21354.975} C_VEL
LIN {X 0,Y 211.041,Z 735.182,A -85,B 0,C 180,E1 -21357.251,E2 -21357.251} C_VEL
LIN {X 0,Y 214.04,Z 725.243,A -85,B 0,C 180,E1 -21359.236,E2 -21359.236} C_VEL
LIN {X 0,Y 216.902,Z 714.201,A -85,B 0,C 180,E1 -21360.955,E2 -21360.955} C_VEL
LIN {X 0,Y 219.551,Z 701.831,A -85,B 0,C 180,E1 -21362.423,E2 -21362.423} C_VEL
LIN {X 0,Y 221.66,Z 689.112,A -85,B 0,C 180,E1 -21363.496,E2 -21363.496} C_VEL
LIN {X 0,Y 223.263,Z 675.674,A -85,B 0,C 180,E1 -21364.24,E2 -21364.24} C_VEL
LIN {X 0,Y 225.462,Z 631.573,A -85,B 0,C 180,E1 -21365.616,E2 -21365.616} C_VEL
LIN {X 0,Y 226.002,Z 617.793,A -85,B 0,C 180,E1 -21366.048,E2 -21366.048} C_VEL
LIN {X 0,Y 223.551,Z 591.907,A -85,B 0,C 180,E1 -21367.552,E2 -21367.552} C_VEL
LIN {X 0,Y 222.417,Z 583.512,A -85,B 0,C 180,E1 -21368.124,E2 -21368.124} C_VEL
LIN {X 0,Y 215.207,Z 564.65,A -85,B 0,C 180,E1 -21370.509,E2 -21370.509} C_VEL
LIN {X 0,Y 212.124,Z 559.455,A -85,B 0,C 180,E1 -21371.479,E2 -21371.479} C_VEL
LIN {X 0,Y 210.916,Z 557.374,A -85,B 0,C 180,E1 -21371.931,E2 -21371.931} C_VEL
LIN {X 0,Y 205.669,Z 546.614,A -85,B 0,C 180,E1 -21375.533,E2 -21375.533} C_VEL
LIN {X 0,Y 201.629,Z 538.71,A -85,B 0,C 180,E1 -21378.527,E2 -21378.527} C_VEL
LIN {X 0,Y 200.235,Z 536.656,A -85,B 0,C 180,E1 -21379.509,E2 -21379.509} C_VEL
LIN {X 0,Y 199.671,Z 534.612,A -85,B 0,C 180,E1 -21380.278,E2 -21380.278} C_VEL
LIN {X 0,Y 199.657,Z 534.596,A -85,B 0,C 180,E1 -21384.056,E2 -21384.056} C_VEL
LIN {X 0,Y 199.701,Z 534.588,A -85,B 0,C 180,E1 -21388.137,E2 -21388.137} C_VEL
LIN {X 0,Y 199.683,Z 534.611,A -85,B 0,C 180,E1 -21392.772,E2 -21392.772} C_VEL
LIN {X 0,Y 199.71,Z 534.58,A -85,B 0,C 180,E1 -21397.226,E2 -21397.226} C_VEL
LIN {X 0,Y 199.792,Z 534.573,A -85,B 0,C 180,E1 -21401.758,E2 -21401.758} C_VEL
LIN {X 0,Y 199.841,Z 534.574,A -85,B 0,C 180,E1 -21405.749,E2 -21405.749} C_VEL
LIN {X 0,Y 200.066,Z 534.537,A -85,B 0,C 180,E1 -21409.884,E2 -21409.884} C_VEL
LIN {X 0,Y 200.031,Z 534.549,A -85,B 0,C 180,E1 -21413.95,E2 -21413.95} C_VEL
LIN {X 0,Y 200.318,Z 534.508,A -85,B 0,C 180,E1 -21417.99,E2 -21417.99} C_VEL
LIN {X 0,Y 200.475,Z 534.472,A -85,B 0,C 180,E1 -21420,E2 -21420} C_VEL
LIN {X 0,Y 200.027,Z 534.569,A -85,B 0,C 180,E1 -21424.03,E2 -21424.03} C_VEL
LIN {X 0,Y 200.085,Z 534.524,A -85,B 0,C 180,E1 -21428.077,E2 -21428.077} C_VEL
LIN {X 0,Y 199.87,Z 534.589,A -85,B 0,C 180,E1 -21432.18,E2 -21432.18} C_VEL
LIN {X 0,Y 199.799,Z 534.563,A -85,B 0,C 180,E1 -21436.345,E2 -21436.345} C_VEL
LIN {X 0,Y 199.821,Z 534.579,A -85,B 0,C 180,E1 -21438.455,E2 -21438.455} C_VEL
LIN {X 0,Y 199.734,Z 534.578,A -85,B 0,C 180,E1 -21443.818,E2 -21443.818} C_VEL
LIN {X 0,Y 199.711,Z 534.59,A -85,B 0,C 180,E1 -21448.388,E2 -21448.388} C_VEL
LIN {X 0,Y 199.676,Z 534.614,A -85,B 0,C 180,E1 -21452.359,E2 -21452.359} C_VEL
LIN {X 0,Y 199.611,Z 534.681,A -85,B 0,C 180,E1 -21456.387,E2 -21456.387} C_VEL
LIN {X 0,Y 202.616,Z 542.274,A -85,B 0,C 180,E1 -21460.264,E2 -21460.264} C_VEL
LIN {X 0,Y 205.848,Z 550.746,A -85,B 0,C 180,E1 -21464.196,E2 -21464.196} C_VEL
LIN {X 0,Y 206.634,Z 552.748,A -85,B 0,C 180,E1 -21464.978,E2 -21464.978} C_VEL
LIN {X 0,Y 213.568,Z 564.586,A -85,B 0,C 180,E1 -21467.278,E2 -21467.278} C_VEL
LIN {X 0,Y 218.674,Z 574.348,A -85,B 0,C 180,E1 -21468.875,E2 -21468.875} C_VEL
LIN {X 0,Y 224.781,Z 587.726,A -85,B 0,C 180,E1 -21470.713,E2 -21470.713} C_VEL
LIN {X 0,Y 226.638,Z 592.471,A -85,B 0,C 180,E1 -21471.27,E2 -21471.27} C_VEL
LIN {X 0,Y 227.475,Z 598.509,A -85,B 0,C 180,E1 -21471.669,E2 -21471.669} C_VEL
LIN {X 0,Y 224.155,Z 663.964,A -85,B 0,C 180,E1 -21473.647,E2 -21473.647} C_VEL
LIN {X 0,Y 222.875,Z 676.514,A -85,B 0,C 180,E1 -21474.313,E2 -21474.313} C_VEL
LIN {X 0,Y 221.006,Z 689.462,A -85,B 0,C 180,E1 -21475.388,E2 -21475.388} C_VEL
LIN {X 0,Y 218.732,Z 701.282,A -85,B 0,C 180,E1 -21476.726,E2 -21476.726} C_VEL
LIN {X 0,Y 216.177,Z 712.344,A -85,B 0,C 180,E1 -21478.388,E2 -21478.388} C_VEL
LIN {X 0,Y 213.135,Z 722.738,A -85,B 0,C 180,E1 -21480.356,E2 -21480.356} C_VEL
LIN {X 0,Y 210.121,Z 732.131,A -85,B 0,C 180,E1 -21482.62,E2 -21482.62} C_VEL
LIN {X 0,Y 207.416,Z 739.818,A -85,B 0,C 180,E1 -21484.942,E2 -21484.942} C_VEL
LIN {X 0,Y 204.654,Z 747.303,A -85,B 0,C 180,E1 -21487.806,E2 -21487.806} C_VEL
LIN {X 0,Y 202.479,Z 753.303,A -85,B 0,C 180,E1 -21490.747,E2 -21490.747} C_VEL
LIN {X 0,Y 200.528,Z 758.042,A -85,B 0,C 180,E1 -21493.718,E2 -21493.718} C_VEL
LIN {X 0,Y 199.133,Z 761.655,A -85,B 0,C 180,E1 -21496.738,E2 -21496.738} C_VEL
LIN {X 0,Y 198.186,Z 764.253,A -85,B 0,C 180,E1 -21499.787,E2 -21499.787} C_VEL
LIN {X 0,Y 197.746,Z 765.47,A -85,B 0,C 180,E1 -21501.827,E2 -21501.827} C_VEL
LIN {X 0,Y 197.447,Z 766.279,A -85,B 0,C 180,E1 -21503.87,E2 -21503.87} C_VEL
LIN {X 0,Y 197.328,Z 766.658,A -85,B 0,C 180,E1 -21505.915,E2 -21505.915} C_VEL
LIN {X 0,Y 197.299,Z 766.659,A -85,B 0,C 180,E1 -21507.959,E2 -21507.959} C_VEL
LIN {X 0,Y 197.375,Z 766.282,A -85,B 0,C 180,E1 -21510,E2 -21510} C_VEL
LIN {X 0,Y 197.493,Z 765.492,A -85,B 0,C 180,E1 -21512.039,E2 -21512.039} C_VEL
LIN {X 0,Y 197.795,Z 764.284,A -85,B 0,C 180,E1 -21514.075,E2 -21514.075} C_VEL
LIN {X 0,Y 198.454,Z 761.399,A -85,B 0,C 180,E1 -21517.431,E2 -21517.431} C_VEL
LIN {X 0,Y 199.769,Z 756.733,A -85,B 0,C 180,E1 -21521.156,E2 -21521.156} C_VEL
LIN {X 0,Y 201.332,Z 751.647,A -85,B 0,C 180,E1 -21524.143,E2 -21524.143} C_VEL
LIN {X 0,Y 203.358,Z 745.24,A -85,B 0,C 180,E1 -21527.083,E2 -21527.083} C_VEL
LIN {X 0,Y 205.861,Z 737.268,A -85,B 0,C 180,E1 -21529.961,E2 -21529.961} C_VEL
LIN {X 0,Y 208.266,Z 729.111,A -85,B 0,C 180,E1 -21532.31,E2 -21532.31} C_VEL
LIN {X 0,Y 210.657,Z 720.207,A -85,B 0,C 180,E1 -21534.384,E2 -21534.384} C_VEL
LIN {X 0,Y 213.382,Z 709.165,A -85,B 0,C 180,E1 -21536.4,E2 -21536.4} C_VEL
LIN {X 0,Y 215.726,Z 697.479,A -85,B 0,C 180,E1 -21538.066,E2 -21538.066} C_VEL
LIN {X 0,Y 217.633,Z 685.75,A -85,B 0,C 180,E1 -21539.317,E2 -21539.317} C_VEL
LIN {X 0,Y 219.069,Z 673.126,A -85,B 0,C 180,E1 -21540.296,E2 -21540.296} C_VEL
LIN {X 0,Y 220.118,Z 659.718,A -85,B 0,C 180,E1 -21540.946,E2 -21540.946} C_VEL
LIN {X 0,Y 223.058,Z 595.992,A -85,B 0,C 180,E1 -21542.879,E2 -21542.879} C_VEL
LIN {X 0,Y 221.444,Z 585.163,A -85,B 0,C 180,E1 -21543.58,E2 -21543.58} C_VEL
LIN {X 0,Y 216.469,Z 573.043,A -85,B 0,C 180,E1 -21544.983,E2 -21544.983} C_VEL
LIN {X 0,Y 209.918,Z 559.731,A -85,B 0,C 180,E1 -21546.863,E2 -21546.863} C_VEL
LIN {X 0,Y 205.908,Z 552.223,A -85,B 0,C 180,E1 -21548.079,E2 -21548.079} C_VEL
LIN {X 0,Y 203.175,Z 544.054,A -85,B 0,C 180,E1 -21551.379,E2 -21551.379} C_VEL
LIN {X 0,Y 201.312,Z 539.299,A -85,B 0,C 180,E1 -21553.465,E2 -21553.465} C_VEL
LIN {X 0,Y 201.197,Z 539.307,A -85,B 0,C 180,E1 -21553.586,E2 -21553.586} C_VEL
LIN {X 0,Y 210.717,Z 567.101,A -85,B 0,C 180,E1 -21555.834,E2 -21555.834} C_VEL
LIN {X 0,Y 207.473,Z 630.038,A -85,B 0,C 180,E1 -21558.98,E2 -21558.98} C_VEL
LIN {X 0,Y 206.639,Z 643.918,A -85,B 0,C 180,E1 -21560.061,E2 -21560.061} C_VEL
LIN {X 0,Y 205.341,Z 657.246,A -85,B 0,C 180,E1 -21561.501,E2 -21561.501} C_VEL
LIN {X 0,Y 204.018,Z 669.425,A -85,B 0,C 180,E1 -21563.234,E2 -21563.234} C_VEL
LIN {X 0,Y 202.607,Z 681.287,A -85,B 0,C 180,E1 -21565.387,E2 -21565.387} C_VEL
LIN {X 0,Y 201.169,Z 692.194,A -85,B 0,C 180,E1 -21567.861,E2 -21567.861} C_VEL
LIN {X 0,Y 199.96,Z 701.673,A -85,B 0,C 180,E1 -21570.523,E2 -21570.523} C_VEL
LIN {X 0,Y 199.058,Z 709.572,A -85,B 0,C 180,E1 -21573.246,E2 -21573.246} C_VEL
LIN {X 0,Y 198.273,Z 717.222,A -85,B 0,C 180,E1 -21576.498,E2 -21576.498} C_VEL
LIN {X 0,Y 197.85,Z 722.308,A -85,B 0,C 180,E1 -21579.193,E2 -21579.193} C_VEL
LIN {X 0,Y 197.626,Z 727.135,A -85,B 0,C 180,E1 -21582.405,E2 -21582.405} C_VEL
LIN {X 0,Y 197.842,Z 730.737,A -85,B 0,C 180,E1 -21585.601,E2 -21585.601} C_VEL
LIN {X 0,Y 198.188,Z 732.519,A -85,B 0,C 180,E1 -21587.715,E2 -21587.715} C_VEL
LIN {X 0,Y 199.209,Z 734.434,A -85,B 0,C 180,E1 -21591.041,E2 -21591.041} C_VEL
LIN {X 0,Y 200.461,Z 735.242,A -85,B 0,C 180,E1 -21593.962,E2 -21593.962} C_VEL
LIN {X 0,Y 201.639,Z 735.27,A -85,B 0,C 180,E1 -21596.002,E2 -21596.002} C_VEL
LIN {X 0,Y 204.642,Z 734.13,A -85,B 0,C 180,E1 -21600,E2 -21600} C_VEL
LIN {X 0,Y 206.463,Z 732.908,A -85,B 0,C 180,E1 -21601.95,E2 -21601.95} C_VEL
LIN {X 0,Y 210.788,Z 729.171,A -85,B 0,C 180,E1 -21605.74,E2 -21605.74} C_VEL
LIN {X 0,Y 214.555,Z 725.169,A -85,B 0,C 180,E1 -21608.476,E2 -21608.476} C_VEL
LIN {X 0,Y 219.436,Z 719.211,A -85,B 0,C 180,E1 -21611.424,E2 -21611.424} C_VEL
LIN {X 0,Y 224.654,Z 711.967,A -85,B 0,C 180,E1 -21614.124,E2 -21614.124} C_VEL
LIN {X 0,Y 229.655,Z 703.933,A -85,B 0,C 180,E1 -21616.443,E2 -21616.443} C_VEL
LIN {X 0,Y 231.134,Z 701.33,A -85,B 0,C 180,E1 -21617.065,E2 -21617.065} C_VEL
LIN {X 0,Y 232.209,Z 698.839,A -85,B 0,C 180,E1 -21617.796,E2 -21617.796} C_VEL
LIN {X 0,Y 233.292,Z 691.627,A -85,B 0,C 180,E1 -21620.603,E2 -21620.603} C_VEL
LIN {X 0,Y 234.395,Z 688.815,A -85,B 0,C 180,E1 -21621.23,E2 -21621.23} C_VEL
LIN {X 0,Y 239.472,Z 677.677,A -85,B 0,C 180,E1 -21622.883,E2 -21622.883} C_VEL
LIN {X 0,Y 243.875,Z 665.943,A -85,B 0,C 180,E1 -21624.246,E2 -21624.246} C_VEL
LIN {X 0,Y 247.496,Z 653.726,A -85,B 0,C 180,E1 -21625.334,E2 -21625.334} C_VEL
LIN {X 0,Y 250.654,Z 639.88,A -85,B 0,C 180,E1 -21626.251,E2 -21626.251} C_VEL
LIN {X 0,Y 255.415,Z 611.864,A -85,B 0,C 180,E1 -21627.523,E2 -21627.523} C_VEL
LIN {X 0,Y 253.923,Z 609.176,A -85,B 0,C 180,E1 -21629.302,E2 -21629.302} C_VEL
LIN {X 0,Y 252.712,Z 607.307,A -85,B 0,C 180,E1 -21631.084,E2 -21631.084} C_VEL
LIN {X 0,Y 251.461,Z 605.932,A -85,B 0,C 180,E1 -21633.985,E2 -21633.985} C_VEL
